# B&R Automation Studio project CControl_Gschneitner (part 5)

#### fbLascoSrvcInterv.st - Funktionsbaustein für Serviceintervalle
```iecst
(********************************************************************
 * COPYRIGHT -- LASCO Heu- und Forsttechnik GmbH
 ********************************************************************
 * Library: LascoUtil
 * Datei: fbLascoSrvcInterv.st
 * Autor: Rudolf Lachner
 * Erstellt: 16. Januar 2014
 ********************************************************************
 * Implementierung der Library LascoUtil
 ********************************************************************)

(* Funktionsbaustein für Serviceintervalle *)
FUNCTION_BLOCK fbLascoSrvcInterv

	//Service rücksetzen
	IF (EDGEPOS(SrvcReset)) THEN
		ZeitBisSrvc	:= SrvcIntervall;
	END_IF

	//Restzeit Countdown
	IF (Aktiv AND Tick) AND (ZeitBisSrvc > 0) THEN
		ZeitBisSrvc	:= ZeitBisSrvc - 1;
	END_IF

	//Service erforderlich
	IF (ZeitBisSrvc = 0) THEN
		SrvcErforderl	:= TRUE;
	ELSE
		SrvcErforderl	:= FALSE;
	END_IF

END_FUNCTION_BLOCK
```

#### fbLascoLstRamp.st - Rampenfunktion, Leistungsanstieg pro Minute
```iecst
(********************************************************************
 * COPYRIGHT -- LASCO Heu- und Forsttechnik GmbH
 ********************************************************************
 * Library: LascoUtil
 * Datei: fbLascoLstRamp.st
 * Autor: Rudolf Lachner
 * Erstellt: 21. Januar 2014
 ********************************************************************
 * Implementierung der Library LascoUtil
 ********************************************************************)

(* Rampenfunktion, Leistungsanstieg pro Minute *)
FUNCTION_BLOCK fbLascoLstRamp

	IF (EDGE(Enable)) THEN
		Fertig			:= FALSE;
		LeistungOut		:= LeistungStart;

	ELSIF (Enable AND sekTick) THEN

		AnstiegProSekunde	:= AnstiegProMinute / 60;

		IF ((LeistungOut + AnstiegProSekunde) <= LeistungSoll) AND NOT Pause THEN
			LeistungOut		:= LeistungOut + AnstiegProSekunde;
		ELSIF ((LeistungOut + AnstiegProSekunde) >= LeistungSoll) AND NOT Pause THEN
			IF LeistungSoll > LeistungStart THEN
				LeistungOut		:= LeistungSoll;
			ELSE
				LeistungOut		:= LeistungStart;
			END_IF
			Fertig 			:= TRUE;
		END_IF
	END_IF

END_FUNCTION_BLOCK
```

#### fbLascoBsk.st - Funktionsbaustein zur Ansteuerung von federrückgestellten Klappenantrieben
```iecst
(********************************************************************
 * COPYRIGHT -- LASCO Heu- und Forsttechnik GmbH
 ********************************************************************
 * Library: LascoUtil
 * Datei: fbLascoBsk.st
 * Autor: rlachner
 * Erstellt: 25. November 2014
 ********************************************************************
 * Implementierung der Library LascoUtil
 ********************************************************************)

(* Funktionsbaustein zur Ansteuerung von federrückgestellten Klappenantrieben *)
FUNCTION_BLOCK fbLascoBsk

	IF Freigabe THEN

		//Fahrzeiten überwachen
		TON_FahrzeitAuf(IN:= KlappeAuf AND NOT KlappeIstOffen AND NOT QuitFehler, PT:= FahrzeitAuf);
		TON_FahrzeitZu(IN:= NOT KlappeAuf AND NOT KlappeIstGeschlossen AND NOT QuitFehler, PT:= FahrzeitZu);

		FehlerFahrzeitAuf	:= TON_FahrzeitAuf.Q;
		FehlerFahrzeitZu	:= TON_FahrzeitZu.Q;

		//Stoerung Absicherung oder Endlagen
		IF (Stoerung) OR (KlappeIstOffen AND KlappeIstGeschlossen) THEN
			Fehler	:= TRUE;
		ELSE
			Fehler	:= FALSE;
		END_IF

		//Fehler rücksetzen
		IF (QuitFehler) THEN
			Fehler				:= FALSE;
		END_IF

		//Ansteuerung Klappe
		KlappeAuf	:= Oeffnen AND NOT Fehler;

	ELSE

		KlappeAuf			:= FALSE;
		Fehler				:= FALSE;
		FehlerFahrzeitAuf	:= FALSE;
		FehlerFahrzeitZu	:= FALSE;
		TON_FahrzeitAuf		(IN:= FALSE);
		TON_FahrzeitZu		(IN:= FALSE);

	END_IF

END_FUNCTION_BLOCK
```

#### fbLascoTrend.st - Trenderkennung eines Eingangswertes innerhalb einer Zeitspanne (steigend/fallend)
```iecst
(********************************************************************
 * COPYRIGHT -- LASCO Heu- und Forsttechnik GmbH
 ********************************************************************
 * Library: LascoUtil
 * Datei: fbLascoTrend.st
 * Autor: Rudolf Lachner
 * Erstellt: 3. Dezember 2014
 ********************************************************************
 * Implementierung der Library LascoUtil
 ********************************************************************)

(* Trenderkennung eines Eingangswertes innerhalb einer Zeitspanne (steigend/fallend) *)
FUNCTION_BLOCK fbLascoTrend

	IF (Freigabe AND (Zeitspanne <> 0)) THEN

		//Mittelwert neu berechnen
		IF (ctZeitspanne >= Zeitspanne) THEN

			Mittelwert	:= ((LREAL_TO_REAL(SummeWert)) / ctZeitspanne);

			//Berechnung der Abweichung
			IF Mittelwert - MittelwertMEM <> 0 THEN
				Abweichung := (((Mittelwert - MittelwertMEM) * 100 ) / ctZeitspanne);
			ELSE
				Abweichung := 0.0;
			END_IF

			//Steigende Tendenz erkannt
			IF MittelwertMEM < (Mittelwert - MinAbweichung) THEN
				TendenzSteigend := TRUE;
			ELSE
				TendenzSteigend := FALSE;
			END_IF

			//Fallende Tendenz erkannt
			IF MittelwertMEM > (Mittelwert + MinAbweichung) THEN
				TendenzFallend := TRUE;
			ELSE
				TendenzFallend := FALSE;
			END_IF

			MittelwertMEM	:= Mittelwert;
			ctZeitspanne	:= 0.0;
			SummeWert		:= 0.0;

		ELSIF Tick THEN

			SummeWert 		:=  SummeWert + Eingangswert;
			ctZeitspanne 	:= ctZeitspanne + 1;

		END_IF

	ELSE

		Abweichung		:= 0.0;
		ctZeitspanne	:= 0.0;
		Mittelwert		:= 0.0;
		MittelwertMEM	:= 0.0;
		SummeWert		:= 0.0;
		TendenzSteigend	:= FALSE;
		TendenzFallend	:= FALSE;

	END_IF

END_FUNCTION_BLOCK
```

#### fbLascoTimerHand.st - Timer mit Hand-Funktionen
```iecst
(********************************************************************
 * COPYRIGHT -- LASCO Heu- und Forsttechnik GmbH
 ********************************************************************
 * Library: LascoUtil
 * Datei: fbLascoTimerHand.st
 * Autor: Rudolf Lachner
 * Erstellt: 9. Dezember 2014
 ********************************************************************
 * Implementierung der Library LascoUtil
 ********************************************************************)

(* Timer mit Hand-Funktionen *)
FUNCTION_BLOCK fbLascoTimerHand

	IF (NOT Freigabe) THEN
		Elapsed	:= 0;
		Q		:= FALSE;
	ELSIF (HandEin) THEN
		Q		:= TRUE;
	ELSIF (HandAus) THEN
		Q		:= FALSE;
	ELSIF (Elapsed >= Zeit) THEN
		Q		:= FALSE;
	ELSE
		Elapsed	:= Elapsed + Tick;
		Q		:= TRUE;
	END_IF

END_FUNCTION_BLOCK
```

#### fbLascoBskUeberw.st - Ansteuerung Brandschutzklappe mit Laufzeitüberwachung und Freiräumung
```iecst
(********************************************************************
 * COPYRIGHT -- Lasco Heutechnik GmbH
 ********************************************************************
 * Library: LascoUtil
 * Datei: fbLascoBskUeberw.st
 * Autor: Rudolf Lachner
 * Erstellt: 20. Juli 2017
 ********************************************************************
 * Implementierung der Library LascoUtil
 ********************************************************************)

(* Ansteuerung Brandschutzklappe mit Laufzeitüberwachung und Freiräumung *)
FUNCTION_BLOCK fbLascoBskUeberw

	//Freigabe
	IF Freigabe THEN

		curStep	:= nextStep;

		//Schrittschaltwerk Überwachung Brandschutzklappe
		//***********************************************

		CASE curStep OF

			//*************************************************************************************************************************************************************************************************************************************
			BSK_WARTEN:

				//*** state entry ***
				IF stateEntry THEN
					stateEntry	:= FALSE;
					TON_Laufzeit(IN	:= FALSE, PT := T#0s);
				END_IF

				//*** state during ***
				//Warten auf Anforderung öffnen oder schließen

				//Fehlerquittierung
				IF Quit THEN
					ctVersucheAuf	:= 0;
					ctVersucheZu	:= 0;
				END_IF

				//*** state exit ***
				//Anforderung Öffnen
				IF FreigabeOeffnen AND NOT loc_KlappeIstOffen THEN
					stateEntry			:= TRUE;
					TON_Laufzeit(IN		:= FALSE, PT := T#0s);
					lastStep			:= curStep;
					nextStep			:= BSK_OEFFNEN;
				//Anforderung Schließen
				ELSIF FreigabeSchliessen AND NOT loc_KlappeIstGeschlossen THEN
					stateEntry			:= TRUE;
					TON_Laufzeit(IN		:= FALSE, PT := T#0s);
					lastStep			:= curStep;
					nextStep			:= BSK_SCHLIESSEN;
				END_IF

			//*************************************************************************************************************************************************************************************************************************************
			BSK_OEFFNEN:

				//*** state entry ***
				IF stateEntry THEN
					stateEntry					:= FALSE;
					TON_Laufzeit(IN				:= FALSE, PT := T#0s);
					loc_KlappeIstGeschlossen	:= FALSE;
					loc_KlappeIstOffen			:= FALSE;
					doKlappeOeffnen				:= TRUE;
				END_IF

				//*** state during ***

				//Laufzeit überwachen
				TON_Laufzeit(IN:= TRUE, PT := LaufzeitAuf);

				//*** state exit ***

				//Klappe ist offen
				IF diKlappeGeoeffnet AND NOT TON_Laufzeit.Q THEN
					TON_Laufzeit(IN		:= FALSE, PT := T#0s);
					ctVersucheAuf		:= 0;
					stateEntry			:= TRUE;
					lastStep			:= curStep;
					nextStep			:= BSK_WARTEN;
					loc_KlappeIstOffen	:= TRUE;

				//Laufzeitüberwachung ausggelöst
				ELSIF TON_Laufzeit.Q THEN
					//Max. Versuche überschritten -> Fehler
					IF ctVersucheAuf >= MaxVersucheAuf THEN
						TON_Laufzeit(IN		:= FALSE, PT := T#0s);
						stateEntry			:= TRUE;
						ctVersucheAuf		:= 0;
						lastStep			:= curStep;
						doKlappeOeffnen		:= FALSE;
						nextStep			:= BSK_STOERUNG;
					//Nächsten Versuch starten
					ELSE
						TON_Laufzeit(IN		:= FALSE, PT := T#0s);
						stateEntry			:= TRUE;
						ctVersucheAuf		:= ctVersucheAuf + 1;
						lastStep			:= curStep;
						doKlappeOeffnen		:= FALSE;
						nextStep			:= BSK_OEFFNEN_FEHLER;
					END_IF
				//Keine Anforderung
				ELSIF NOT FreigabeOeffnen THEN
					TON_Laufzeit(IN			:= FALSE, PT := T#0s);
					ctVersucheAuf			:= 0;
					stateEntry				:= TRUE;
					lastStep				:= curStep;
					nextStep				:= BSK_WARTEN;
				END_IF

			//*************************************************************************************************************************************************************************************************************************************
			BSK_OEFFNEN_FEHLER:

				//*** state entry ***
				IF stateEntry THEN
					stateEntry			:= FALSE;
					TON_Laufzeit(IN		:= FALSE, PT := T#0s);
				END_IF

				//*** state during ***

				//Laufzeit überwachen
				TON_Laufzeit(IN:= TRUE, PT := LaufzeitZu);

				//*** state exit ***
				//Klappe geschlossen -> Versuch öffnen
				IF diKlappeGeschlossen AND FreigabeOeffnen THEN
					stateEntry			:= TRUE;
					ctVersucheZu		:= 0;
					lastStep			:= curStep;
					nextStep			:= BSK_OEFFNEN;
					TON_Laufzeit(IN		:= FALSE, PT := T#0s);
				//Laufzeit überschritten
				ELSIF TON_Laufzeit.Q THEN
					//Max. Versuche überschritten -> Fehler
					IF ctVersucheZu >= MaxVersucheZu THEN
						TON_Laufzeit(IN		:= FALSE, PT := T#0s);
						stateEntry			:= TRUE;
						ctVersucheZu		:= 0;
						lastStep			:= curStep;
						doKlappeOeffnen		:= FALSE;
						nextStep			:= BSK_STOERUNG;
					//Nächsten Versuch starten
					ELSE
						TON_Laufzeit(IN		:= FALSE, PT := T#0s);
						stateEntry			:= TRUE;
						ctVersucheZu		:= ctVersucheZu + 1;
						lastStep			:= curStep;
						nextStep			:= BSK_OEFFNEN;
					END_IF
				//Keine Freigabe Öffnen
				ELSIF NOT FreigabeOeffnen THEN
					stateEntry				:= TRUE;
					TON_Laufzeit(IN			:= FALSE, PT := T#0s);
					lastStep				:= curStep;
					ctVersucheAuf			:= 0;
					nextStep				:= BSK_WARTEN;
				END_IF

			//*************************************************************************************************************************************************************************************************************************************
			BSK_SCHLIESSEN:

				//*** state entry ***
				IF stateEntry THEN
					stateEntry					:= FALSE;
					TON_Laufzeit(IN				:= FALSE, PT := T#0s);
					loc_KlappeIstGeschlossen	:= FALSE;
					loc_KlappeIstOffen			:= FALSE;
					doKlappeOeffnen				:= FALSE;
				END_IF

				//*** state during ***

				//Laufzeit überwachen
				TON_Laufzeit(IN:= TRUE, PT := LaufzeitZu);

				//*** state exit ***

				//Klappe ist geschlossen
				IF diKlappeGeschlossen AND NOT TON_Laufzeit.Q THEN
					TON_Laufzeit(IN				:= FALSE, PT := T#0s);
					ctVersucheZu				:= 0;
					stateEntry					:= TRUE;
					lastStep					:= curStep;
					nextStep					:= BSK_WARTEN;
					loc_KlappeIstGeschlossen	:= TRUE;

					//Laufzeitüberwachung ausgelöst
				ELSIF TON_Laufzeit.Q THEN
					//Max. Versuche überschritten -> Fehler
					IF ctVersucheZu >= MaxVersucheZu THEN
						TON_Laufzeit(IN		:= FALSE, PT := T#0s);
						stateEntry			:= TRUE;
						ctVersucheZu		:= 0;
						lastStep			:= curStep;
						doKlappeOeffnen		:= FALSE;
						nextStep			:= BSK_STOERUNG;
					//Nächsten Versuch starten
					ELSE
						TON_Laufzeit(IN		:= FALSE, PT := T#0s);
						stateEntry			:= TRUE;
						ctVersucheZu		:= ctVersucheZu + 1;
						lastStep			:= curStep;
						nextStep			:= BSK_SCHLIESSEN_FEHLER;
					END_IF
				//Anforderung Oeffnen
				ELSIF  FreigabeOeffnen THEN
					TON_Laufzeit(IN			:= FALSE, PT := T#0s);
					ctVersucheZu			:= 0;
					stateEntry				:= TRUE;
					lastStep				:= curStep;
					nextStep				:= BSK_WARTEN;
				END_IF

			//*************************************************************************************************************************************************************************************************************************************
			BSK_SCHLIESSEN_FEHLER:

				//*** state entry ***
				IF stateEntry THEN
					stateEntry			:= FALSE;
					TON_Laufzeit(IN		:= FALSE, PT := T#0s);
					doKlappeOeffnen		:= TRUE;
				END_IF

				//*** state during ***

				//Laufzeit überwachen
				TON_Laufzeit(IN:= TRUE, PT := LaufzeitAuf);

				//*** state exit ***
				//Klappe offen -> Versuch schließen
				IF diKlappeGeoeffnet AND FreigabeSchliessen THEN
					stateEntry			:= TRUE;
					ctVersucheAuf		:= 0;
					lastStep			:= curStep;
					nextStep			:= BSK_SCHLIESSEN;
					TON_Laufzeit(IN		:= FALSE, PT := T#0s);
				//Laufzeit überschritten
				ELSIF TON_Laufzeit.Q THEN
					//Max. Versuche überschritten -> Fehler
					IF ctVersucheAuf >= MaxVersucheAuf THEN
						TON_Laufzeit(IN		:= FALSE, PT := T#0s);
						stateEntry			:= TRUE;
						ctVersucheAuf		:= 0;
						lastStep			:= curStep;
						doKlappeOeffnen		:= FALSE;
						nextStep			:= BSK_STOERUNG;
						//Nächsten Versuch starten
					ELSE
						TON_Laufzeit(IN		:= FALSE, PT := T#0s);
						stateEntry			:= TRUE;
						ctVersucheAuf		:= ctVersucheAuf + 1;
						lastStep			:= curStep;
						nextStep			:= BSK_SCHLIESSEN;
					END_IF
					//Freigabe Öffnen
				ELSIF FreigabeOeffnen THEN
					stateEntry				:= TRUE;
					TON_Laufzeit(IN			:= FALSE, PT := T#0s);
					lastStep				:= curStep;
					ctVersucheZu			:= 0;
					nextStep				:= BSK_WARTEN;
				END_IF

			//*************************************************************************************************************************************************************************************************************************************
			BSK_STOERUNG:

				//*** state entry ***
				IF stateEntry THEN
					stateEntry		:= FALSE;
					TON_Laufzeit(IN	:= FALSE, PT := T#0s);
					Stoerung		:= TRUE;
				END_IF

				//*** state during ***
				//Warten auf Quittierung

				//*** state exit ***
				IF Quit THEN
					stateEntry	:= TRUE;
					Stoerung	:= FALSE;
					lastStep	:= curStep;
					nextStep	:= BSK_WARTEN;
				END_IF

		END_CASE

	//Keine Freigabe Funktionsbaustein
	ELSE

		//Alle Parameter zurücksetzen
		doKlappeOeffnen	:= FALSE;
		ctVersucheAuf	:= 0;
		ctVersucheZu	:= 0;
		Stoerung		:= FALSE;
		TON_Laufzeit(IN	:= FALSE, PT := T#0s);
		stateEntry		:= TRUE;
		curStep			:= BSK_WARTEN;
		nextStep		:= BSK_WARTEN;
		lastStep		:= BSK_WARTEN;

	END_IF

END_FUNCTION_BLOCK
```

#### fbLascoAutoRuecklauf.st - Automatische Rücklauffunktion für Motoren
```iecst
(********************************************************************
 * COPYRIGHT -- LASCO Heu- und Forsttechnik GmbH
 ********************************************************************
 * Library: LascoUtil
 * Datei: fbLascoAutoRuecklauf.st
 * Autor: rlachner
 * Erstellt: 24. Februar 2014
 ********************************************************************
 * Implementierung der Library LascoUtil
 ********************************************************************)

(* Automatische Rücklauffunktion für Motoren *)
FUNCTION_BLOCK fbLascoAutoRuecklauf

	IF Freigabe THEN

		CASE loc_curStep OF

			//AUS ********************************************************************************************************
			0:

				IF stateEntry THEN
					stateEntry := FALSE;
				END_IF

				MotorVor	:= FALSE;
				MotorRueck	:= FALSE;

				IF Zuendphase THEN
					stateEntry		:= TRUE;
					loc_curStep		:= 1;
				ELSIF Heizphase THEN
					stateEntry		:= TRUE;
					loc_curStep		:= 3;
				END_IF

			//ZUENDPHASE ***************************************************************************************************
			1:

				IF stateEntry THEN
					stateEntry 				:= FALSE;
					ctLaufzeitEinschub1		:= 0;
					ctLaufzeitEinschubVor	:= 0;
				END_IF

				MotorVor				:= (LaufzeitEinschubZuendung >= ctLaufzeitEinschub1);

				//Gesamtlaufzeit Motor Vor
				IF (ctLaufzeitEinschub1 <= LaufzeitEinschubZuendung) THEN
					ctLaufzeitEinschub1	:= ctLaufzeitEinschub1 + sekTick;
				END_IF

				//Laufzeit Vor am Stück
				IF MotorVor THEN
					ctLaufzeitEinschubVor	:= ctLaufzeitEinschubVor + sekTick;
				END_IF

				//Rücklauf erforderlich
				IF (ctLaufzeitEinschubVor >= MaxLaufzeitVor) AND (ctLaufzeitEinschub1 < LaufzeitEinschubZuendung) THEN
					loc_RuecklaufErforderlich	:= TRUE;
				END_IF

				//*** state exit ***
				IF (NOT Zuendphase) THEN
					stateEntry	:= TRUE;
					loc_curStep	:= 0;
				ELSIF loc_RuecklaufErforderlich THEN
					ctLaufzeitEinschubVor	:= 0;
					stateEntry	:= TRUE;
					loc_curStep	:= 2;
				END_IF

			//Zuendphase= Motor zurück ************************************************************************************************************
			2:

				IF stateEntry THEN
					stateEntry 				:= FALSE;
					MotorVor				:= FALSE;
					TON_Umschaltverz.IN		:= TRUE;
				END_IF

				TON_Umschaltverz.PT			:= VerzUmschaltung;
				TON_Umschaltverz();

				TOF_Ruecklauf.IN			:= TON_Umschaltverz.Q AND loc_RuecklaufErforderlich;
				TOF_Ruecklauf.PT			:= Ruecklaufzeit;
				TOF_Ruecklauf();

				MotorRueck					:= TOF_Ruecklauf.Q;

				IF MotorRueck THEN
					loc_RuecklaufErforderlich	:= FALSE;
				END_IF

				IF EDGENEG(MotorRueck) THEN
					loc_RueckwaertsOk	:= TRUE;
					TON_Umschaltverz(IN:= FALSE);
					TON_Umschaltverz.IN	:= TRUE;
				END_IF

				IF TON_Umschaltverz.Q AND loc_RueckwaertsOk THEN
					loc_RueckwaertsOk	:= FALSE;
					loc_curStep	:= 1;
					TON_Umschaltverz(IN:= FALSE);
					TOF_Ruecklauf(IN:= FALSE);
				ELSIF NOT Zuendphase THEN
					loc_curStep	:= 0;
					stateEntry	:= TRUE;
				END_IF

			//Heizphase ************************************************************************************************************
			3:

				//Vorwärts- Impulse mitzählen
				IF (EDGEPOS(ImpulsVor)) THEN
					ctEinschuebeSeitRuecklauf	:= ctEinschuebeSeitRuecklauf + 1;
				ELSIF (MotorRueck) THEN
					ctEinschuebeSeitRuecklauf	:= 0;
				END_IF

				//Kommando Rückwärtsfahrt erforderlich
				IF (ctEinschuebeSeitRuecklauf >= ImpulseVorBisRueck) AND NOT (ImpulsVor) THEN
					loc_RuecklaufErforderlich	:= TRUE;
				ELSIF (MotorRueck) THEN
					loc_RuecklaufErforderlich	:= FALSE;
				END_IF

				//Umschaltverzögerung
				IF (EDGENEG(ImpulsVor)) AND (loc_RuecklaufErforderlich) THEN
					TON_Umschaltverz.IN			:= TRUE;
				ELSIF (EDGEPOS(ImpulsVor)) THEN
					TON_Umschaltverz.IN			:= FALSE;
				END_IF

				//Rücklaufzeit
				TOF_Ruecklauf.IN	:= loc_RuecklaufErforderlich AND TON_Umschaltverz.Q;

				//Kommando "Motor Rückwärts"
				MotorRueck			:= TOF_Ruecklauf.Q;

				//Timer aufrufen
				TON_Umschaltverz.PT	:= UDINT_TO_TIME(VerzUmschaltung);
				TON_Umschaltverz();

				TOF_Ruecklauf.PT	:= UDINT_TO_TIME(Ruecklaufzeit);
				TOF_Ruecklauf();

				IF (NOT Heizphase) THEN
					loc_curStep	:= 0;
					stateEntry	:= TRUE;
				END_IF

		END_CASE

	ELSE

		stateEntry					:= TRUE;
		loc_curStep					:= 0;
		ctLaufzeitEinschub1			:= 0;
		ctLaufzeitEinschubVor		:= 0;
		MotorVor					:= FALSE;
		MotorRueck					:= FALSE;
		loc_RuecklaufErforderlich	:= FALSE;
		loc_RueckwaertsOk			:= FALSE;
		ctEinschuebeSeitRuecklauf	:= 0;
		TON_Umschaltverz.IN			:= FALSE;
		TOF_Ruecklauf.IN			:= FALSE;

	END_IF

END_FUNCTION_BLOCK
```

#### fbLascoPugeV2.st
```iecst
(* Puls/Pause-Generator mit Standard-Timern *)
FUNCTION_BLOCK fbLascoPugeV2

	curStep	:= nextStep;

	CASE curStep OF

		//*******************************************************************************************************************************************************************************
		0://WARTEN

			//*** state entry ***
			IF stateEntry THEN
				stateEntry := FALSE;
				PulsOut := FALSE;
				PauseOut := FALSE;
				TON_Schrittzeit(IN:= FALSE);
				RestzeitPause	:= 0;
				RestzeitPuls	:= 0;
			END_IF

			//*** state during ***

			//*** state exit ***
			IF (StartMitPuls) AND (ZeitPuls <> 0) THEN
				stateEntry := TRUE;
				nextStep	:= 2;
			ELSIF (StartMitPause) THEN
				stateEntry := TRUE;
				nextStep	:= 1;
			END_IF

			//***********************************************************************************************************************************************************************************
		1://PAUSE

			//*** state entry ***
			IF stateEntry THEN
				stateEntry := FALSE;
				PulsOut := FALSE;
				PauseOut := TRUE;
				TON_Schrittzeit(IN:= FALSE);
				RestzeitPause	:= 0;
				RestzeitPuls	:= 0;
			END_IF

			//*** state during ***
			TON_Schrittzeit(IN:= TRUE, PT:= UDINT_TO_TIME(ZeitPause));
			RestzeitPause := ZeitPause - TIME_TO_UDINT(TON_Schrittzeit.ET);

			//*** state exit ***
			IF (NOT StartMitPause AND NOT StartMitPuls) OR (ZeitPuls = 0) THEN
				stateEntry := TRUE;
				nextStep := 0;
			ELSIF TON_Schrittzeit.Q THEN
				stateEntry := TRUE;
				nextStep := 2;
			END_IF

			//************************************************************************************************************************************************************************************************
		2://PULS

			//*** state entry ***
			IF stateEntry THEN
				stateEntry := FALSE;
				PulsOut := TRUE;
				PauseOut := FALSE;
				TON_Schrittzeit(IN:= FALSE);
				RestzeitPause	:= 0;
				RestzeitPuls	:= 0;
			END_IF

			//*** state during ***
			TON_Schrittzeit(IN:= TRUE, PT:= UDINT_TO_TIME(ZeitPuls));
			RestzeitPuls := ZeitPuls - TIME_TO_UDINT(TON_Schrittzeit.ET);

			//*** state exit ***
			IF (NOT StartMitPause AND NOT StartMitPuls) OR (ZeitPuls = 0) THEN
				stateEntry := TRUE;
				nextStep := 0;
			ELSIF TON_Schrittzeit.Q THEN
				stateEntry := TRUE;
				nextStep := 1;
			END_IF

	END_CASE

END_FUNCTION_BLOCK
```

### Library Logical/Libraries/LaEntfV2 (IEC, version 1.00.0) - Funktionsblöcke für Entfeuchter ab LaTronicCControl407Plus

#### LaEntfV2.fun - Exported functions and function blocks
```iecst
{REDUND_UNREPLICABLE} FUNCTION_BLOCK fbEntfOelsumpfheiz (*Funktionsbaustein für Ansteuerung Ölsumpfheizung*) (*$GROUP=User,$CAT=User,$GROUPICON=User.png,$CATICON=User.png*)
	VAR_INPUT
		EintrittTemp : {REDUND_UNREPLICABLE} REAL;
		parTempOelsumpfheizungAus : {REDUND_UNREPLICABLE} REAL;
		parTempOelsumpfheizungEin : {REDUND_UNREPLICABLE} REAL;
		Freigabe : {REDUND_UNREPLICABLE} BOOL;
		StatusSensorEintrittOk : {REDUND_UNREPLICABLE} BOOL;
	END_VAR
	VAR_OUTPUT
		OelsumpfheizungEin : {REDUND_UNREPLICABLE} BOOL;
	END_VAR
END_FUNCTION_BLOCK

{REDUND_UNREPLICABLE} FUNCTION_BLOCK fbEntfKompressor (*Funktionsbaustein für Ansteuerung Kompressor*) (*$GROUP=User,$CAT=User,$GROUPICON=User.png,$CATICON=User.png*)
	VAR_INPUT
		EintrittFeuchte : {REDUND_UNREPLICABLE} REAL;
		SicherheitOk : {REDUND_UNREPLICABLE} BOOL;
		Freigabe : {REDUND_UNREPLICABLE} BOOL;
		BetriebsmldgVentilator : {REDUND_UNREPLICABLE} BOOL;
		Automatik : {REDUND_UNREPLICABLE} BOOL;
		Dauerbetrieb : {REDUND_UNREPLICABLE} BOOL;
		parFeuchteEin : {REDUND_UNREPLICABLE} REAL;
		parFeuchteAus : {REDUND_UNREPLICABLE} REAL;
		parEinschaltverzAbtau : {REDUND_UNREPLICABLE} UDINT;
		parAusschaltverzAbtau : {REDUND_UNREPLICABLE} UDINT;
		parEinschaltverzKompressor : {REDUND_UNREPLICABLE} UDINT;
		Hochdruck : {REDUND_UNREPLICABLE} REAL;
		Niederdruck : {REDUND_UNREPLICABLE} REAL;
		parNiederdruckMin : {REDUND_UNREPLICABLE} REAL;
		parHochdruckMax : {REDUND_UNREPLICABLE} REAL;
		parNiederdruckMax : {REDUND_UNREPLICABLE} REAL;
		StatusSensorNiederdruckOk : {REDUND_UNREPLICABLE} BOOL;
		StatusSensorEintrittOk : {REDUND_UNREPLICABLE} BOOL;
		DrehzahlvorgabeFU : {REDUND_UNREPLICABLE} REAL;
		BetriebsmldgKompressor : {REDUND_UNREPLICABLE} BOOL;
		DrehzahlMin : {REDUND_UNREPLICABLE} REAL;
		DrehzahlMax : {REDUND_UNREPLICABLE} REAL;
		RampeUp : {REDUND_UNREPLICABLE} REAL;
		RampeDown : {REDUND_UNREPLICABLE} REAL;
		QuitFehler : {REDUND_UNREPLICABLE} BOOL;
		parEinschaltverzMagnetventil : {REDUND_UNREPLICABLE} UDINT;
		parNiederdruckPumpdown : {REDUND_UNREPLICABLE} REAL;
		diNiederdruckOk : {REDUND_UNREPLICABLE} BOOL;
		diHochdruckOk : {REDUND_UNREPLICABLE} BOOL;
		KlappenumschaltungAkiv : {REDUND_UNREPLICABLE} BOOL;
		parVerzStandbyBeiKlappenumsch : {REDUND_UNREPLICABLE} UDINT;
	END_VAR
	VAR_OUTPUT
		FreigabeKompressorOut : {REDUND_UNREPLICABLE} BOOL;
		StoerungOut : {REDUND_UNREPLICABLE} BOOL;
		AbtauungAktiv : {REDUND_UNREPLICABLE} BOOL;
		DrehzahlOut : {REDUND_UNREPLICABLE} REAL;
		MagnetventilOut : {REDUND_UNREPLICABLE} BOOL;
		curStep : {REDUND_UNREPLICABLE} USINT;
		loc_StatusFeuchteOk : {REDUND_UNREPLICABLE} BOOL;
		FehlerPumpdown : {REDUND_UNREPLICABLE} BOOL;
		StandbyKlappenumsch : {REDUND_UNREPLICABLE} BOOL;
	END_VAR
	VAR
		TON_Abtau : {REDUND_UNREPLICABLE} TON;
		TON_Kompressor : {REDUND_UNREPLICABLE} TON;
		lastStep : {REDUND_UNREPLICABLE} USINT;
		nextStep : {REDUND_UNREPLICABLE} USINT;
		stateEntry : {REDUND_UNREPLICABLE} BOOL;
		fbFuKompressor : {REDUND_UNREPLICABLE} fbLascoFU;
		sekTick : {REDUND_UNREPLICABLE} BOOL;
		fbLascoEUhr_0 : {REDUND_UNREPLICABLE} fbLascoEUhr;
		fbLascoZdxx_0 : {REDUND_UNREPLICABLE} fbLascoZdxx;
		TON_EinschaltverzMagnetventil : {REDUND_UNREPLICABLE} TON;
		TON_LaufzeitPumpdown : {REDUND_UNREPLICABLE} TON;
		TON_Klappenumschaltung : {REDUND_UNREPLICABLE} TON;
	END_VAR
END_FUNCTION_BLOCK

{REDUND_ERROR} {REDUND_UNREPLICABLE} FUNCTION_BLOCK fbEntfFremd (*Funktionsbaustein zur Ansteuerung von Entfeuchtern (Fremdgeräte)*) (*$GROUP=User,$CAT=User,$GROUPICON=User.png,$CATICON=User.png*)
	VAR_INPUT
		Freigabe : {REDUND_UNREPLICABLE} BOOL;
		StoerungIn : {REDUND_UNREPLICABLE} BOOL;
		parVerzStoerung : {REDUND_UNREPLICABLE} UDINT;
		QuitFehler : {REDUND_UNREPLICABLE} BOOL;
		Dauerbetrieb : {REDUND_UNREPLICABLE} BOOL;
		Automatik : {REDUND_UNREPLICABLE} BOOL;
		BetriebsmldgVentilator : {REDUND_UNREPLICABLE} BOOL;
		parEinschaltverzKompressor : {REDUND_UNREPLICABLE} UDINT;
		BetriebsmldgEntfeuchter : {REDUND_UNREPLICABLE} BOOL;
		WitterungIstSchlecht : {REDUND_UNREPLICABLE} BOOL; (*Wenn TRUE, wird der Entfeuchter im Automatikbetrieb freigegeben*)
		parVerzBetriebEntfeuchter : {REDUND_UNREPLICABLE} UDINT;
	END_VAR
	VAR_OUTPUT
		StoerungOut : {REDUND_UNREPLICABLE} BOOL;
		FehlerBetriebsmldg : {REDUND_UNREPLICABLE} BOOL;
		FreigabeKompressorOut : {REDUND_UNREPLICABLE} BOOL;
	END_VAR
	VAR
		TON_Stoerung : {REDUND_UNREPLICABLE} TON;
		TON_VerzBetriebsmeldung : {REDUND_UNREPLICABLE} TON;
		curStep : {REDUND_UNREPLICABLE} USINT;
		nextStep : {REDUND_UNREPLICABLE} USINT;
		stateEntry : {REDUND_UNREPLICABLE} BOOL;
		TON_Kompressor : {REDUND_UNREPLICABLE} TON;
		lastStep : {REDUND_UNREPLICABLE} USINT;
	END_VAR
END_FUNCTION_BLOCK
```

#### fbEntfOelsumpfheiz.st
```iecst
(* Funktionsbaustein für Ansteuerung Oelsumpfheizung *)
FUNCTION_BLOCK fbEntfOelsumpfheiz

	//Ansteuerung Ölsumpfheizung
	//==========================

	IF Freigabe THEN

		OelsumpfheizungEin	:= TRUE;

	ELSE
		OelsumpfheizungEin	:= FALSE;
	END_IF

END_FUNCTION_BLOCK
```

#### fbEntfKompressor.st
```iecst
(* Ansteuerung Kompressor *)
FUNCTION_BLOCK fbEntfKompressor

	//Zeitticks erzeugen
	fbLascoEUhr_0(Freigabe := TRUE);
	fbLascoZdxx_0(IN := fbLascoEUhr_0.Sekunde);
	sekTick	:= fbLascoZdxx_0.Q;

	//Ausgang Störung Ein, wenn Sicherheitskreis nicht ok
	IF NOT SicherheitOk OR (fbFuKompressor.StoerungFU) THEN
		StoerungOut	:= TRUE;
	END_IF

	//Störung Laufzeit Pumpdown zurücksetzen, wenn Fehler quittiert
	IF QuitFehler THEN
		FehlerPumpdown	:= FALSE;
		StoerungOut		:= FALSE;
	END_IF

	//Funktionsbaustein FU Kompressor
	fbFuKompressor.AnsprechZeitFU	:= 5;
	fbFuKompressor.BetrMldg			:= BetriebsmldgKompressor;
	fbFuKompressor.MinDrehzahl		:= 0.0;
	fbFuKompressor.MaxDrehzahl		:= DrehzahlMax;
	fbFuKompressor.RampeUpSek		:= RampeUp;
	fbFuKompressor.RampeDownSek		:= RampeDown;
	fbFuKompressor.Reset			:= QuitFehler;
	fbFuKompressor.Tick				:= sekTick;
	fbFuKompressor();
	FreigabeKompressorOut			:= fbFuKompressor.BetriebFU;
	DrehzahlOut						:= fbFuKompressor.DrehzahlFU;

	//Schaltpunkte für Eintritt Feuchte generieren
	IF NOT Dauerbetrieb AND NOT Automatik THEN
		loc_StatusFeuchteOk := FALSE;
	ELSIF Dauerbetrieb THEN
		loc_StatusFeuchteOk	:= TRUE;
	ELSIF (EintrittFeuchte <= parFeuchteAus) AND loc_StatusFeuchteOk THEN
		loc_StatusFeuchteOk	:= FALSE;
	ELSIF (EintrittFeuchte >= parFeuchteEin) AND NOT loc_StatusFeuchteOk THEN
		loc_StatusFeuchteOk	:= TRUE;
	END_IF

	curStep	:= nextStep;

	CASE curStep OF

		//AUS **************************************************************************************************************************************
		0:

			//*** state entry ***
			IF stateEntry THEN
				stateEntry					:= FALSE;
				fbFuKompressor.Freigabe		:= FALSE;
				fbFuKompressor.SollDrehzahl	:= 0.0;
				TON_EinschaltverzMagnetventil(IN:= FALSE, PT:= 0);
				TON_Kompressor(IN:= FALSE, PT:= 0);
				TON_Abtau(IN:= FALSE, PT:= 0);
				AbtauungAktiv				:= FALSE;
				MagnetventilOut				:= FALSE;
			END_IF

			//*** state during ***
			//Warten auf Freigabe

			//*** state exit ***
			//Automatik oder Dauerbetrieb, Sensoren OK, Sicherheitskreis geschlossen, Ventilator in Betrieb -> Kompressor Ein
			IF ((Automatik AND StatusSensorEintrittOk) OR Dauerbetrieb) AND Freigabe AND StatusSensorNiederdruckOk AND loc_StatusFeuchteOk
				AND SicherheitOk AND BetriebsmldgVentilator AND diHochdruckOk AND diNiederdruckOk THEN
				nextStep	:= 1;
				lastStep	:= curStep;
				stateEntry	:= TRUE;
			ELSE
				nextStep	:= curStep;
			END_IF

		//KOMPRESSOR EIN **************************************************************************************************************************************
		1:

			//*** state entry ***
			IF stateEntry THEN
				stateEntry	:= FALSE;
				TON_Kompressor(IN:= FALSE, PT:= 0);
				fbFuKompressor.Freigabe		:= FALSE;
				fbFuKompressor.SollDrehzahl	:= 0.0;
				MagnetventilOut				:= FALSE;
				AbtauungAktiv				:= FALSE;
			END_IF

			//*** state during ***

			//Einschaltverzögerung Kompressor starten
			TON_Kompressor(IN:= TRUE, PT := parEinschaltverzKompressor);

			fbFuKompressor.Freigabe		:= TON_Kompressor.Q;
			fbFuKompressor.SollDrehzahl	:= DrehzahlvorgabeFU;

			//*** state exit ***
			//Keine Automatik und kein Dauerbetrieb, Sicherheit nicht ok, keine Betriebsmeldung Ventilator
			//oder Status Sensoren nicht ok -> AUS
			IF (NOT Automatik AND NOT Dauerbetrieb) OR (NOT StatusSensorEintrittOk AND Automatik) OR (NOT Freigabe) OR
				(NOT StatusSensorNiederdruckOk) OR (NOT SicherheitOk) OR (NOT BetriebsmldgVentilator) OR (NOT loc_StatusFeuchteOk) OR (NOT diHochdruckOk) OR (NOT diNiederdruckOk) THEN
				stateEntry	:= TRUE;
				lastStep	:= curStep;
				nextStep	:= 0;
			//Kompressor läuft -> Magnetventil Ein
			ELSIF fbFuKompressor.Freigabe THEN
				stateEntry	:= TRUE;
				lastStep	:= curStep;
				nextStep	:= 2;
			END_IF

		//MAGNETVENTIL EIN **************************************************************************************************************************************
		2:

			//*** state entry ***
			IF stateEntry THEN
				stateEntry	:= FALSE;
				TON_Kompressor(IN:= FALSE, PT:= 0);
				TON_EinschaltverzMagnetventil(IN:= FALSE, PT:= 0);
				MagnetventilOut				:= FALSE;
			END_IF

			//*** state during ***

			//Einschaltverzögerung Magnetventil
			TON_EinschaltverzMagnetventil(IN:= TRUE, PT:= parEinschaltverzMagnetventil);
			MagnetventilOut	:= (TON_EinschaltverzMagnetventil.Q) OR (parEinschaltverzMagnetventil = 0);

			//*** state exit ***
			//Keine Automatik und kein Dauerbetrieb, Sicherheit nicht ok, keine Betriebsmeldung Ventilator
			//oder Status Sensoren nicht ok -> Magnetventil Aus
			IF (NOT Automatik AND NOT Dauerbetrieb) OR (NOT StatusSensorEintrittOk AND Automatik) OR (NOT Freigabe) OR
				(NOT StatusSensorNiederdruckOk) OR (NOT SicherheitOk) OR (NOT BetriebsmldgVentilator) OR (NOT diHochdruckOk) OR (NOT diNiederdruckOk)  THEN
				stateEntry	:= TRUE;
				lastStep	:= curStep;
				IF MagnetventilOut THEN
					nextStep	:= 4;
				ELSE
					nextStep	:= 0;
				END_IF
			//Magnetventil Ein -> Betrieb
			ELSIF MagnetventilOut THEN
				stateEntry	:= TRUE;
				lastStep	:= curStep;
				nextStep	:= 3;
			END_IF

		//BETRIEB **************************************************************************************************************************************
		3:

			//*** state entry ***
			IF stateEntry THEN
				stateEntry		:= FALSE;
				TON_Abtau(IN:= FALSE, PT:= 0);
				AbtauungAktiv	:= FALSE;
				TON_Klappenumschaltung(IN:= FALSE, PT:= 0);
			END_IF

			//*** state during ***
			//Kompressor Drehzahlvorgabe
			fbFuKompressor.SollDrehzahl	:= DrehzahlvorgabeFU;

			//Verzöguerung Abtauung starten, wenn Niederdruck unter Min.
			TON_Abtau(IN:= (Niederdruck <= parNiederdruckMin), PT:= parEinschaltverzAbtau);

			//Wenn Hochdruck Max. überschritten & Klappenumschaltung aktiv -> Verzögerung starten für Standby
			TON_Klappenumschaltung(IN:= (Hochdruck > parHochdruckMax) AND KlappenumschaltungAkiv, PT:= parVerzStandbyBeiKlappenumsch);

			//*** state exit ***
			//Keine Automatik und kein Dauerbetrieb, Sicherheit nicht ok, keine Betriebsmeldung Ventilator
			//oder Status Sensoren nicht ok -> Magnetventil Aus
			IF (NOT Automatik AND NOT Dauerbetrieb) OR (NOT StatusSensorEintrittOk AND Automatik) OR (NOT Freigabe) OR
				(NOT StatusSensorNiederdruckOk) OR (NOT SicherheitOk) OR (NOT BetriebsmldgVentilator) OR (NOT loc_StatusFeuchteOk) OR (NOT diHochdruckOk) OR (NOT diNiederdruckOk) THEN
				stateEntry	:= TRUE;
				lastStep	:= curStep;
				nextStep	:= 4;
			//Abtauung angesprochen -> Abtauung
			ELSIF TON_Abtau.Q THEN
				stateEntry		:= TRUE;
				AbtauungAktiv	:= TRUE;
				nextStep		:= 6;
				lastStep		:= curStep;
			//Hochdruck Max. während Klappenumschaltung überschritten -> Standby
			ELSIF TON_Klappenumschaltung.Q THEN
				stateEntry		:= TRUE;
				nextStep		:= 7;
				lastStep		:= curStep;
			ELSE
				nextStep		:= curStep;
			END_IF

		//MAGNETVENTIL AUS **************************************************************************************************************************************
		4:

			//*** state entry ***
			IF stateEntry THEN
				stateEntry		:= FALSE;
				TON_Abtau(IN	:= FALSE, PT:= 0);
				AbtauungAktiv	:= FALSE;
				MagnetventilOut	:= FALSE;
				fbFuKompressor.SollDrehzahl	:= DrehzahlMin;
				TON_LaufzeitPumpdown(IN:= FALSE, PT:= 0);
			END_IF

			//*** state during ***

			//Laufzeit Pumpdown überwachen
			TON_LaufzeitPumpdown(IN:= TRUE, PT:= T#5m);

			//*** state exit ***
			//Automatik oder Dauerbetrieb, Sensoren und Sicherheit ok, Ventilator in Betrieb -> Betrieb
			IF ((Automatik AND StatusSensorEintrittOk) OR Dauerbetrieb) AND StatusSensorNiederdruckOk AND SicherheitOk AND Freigabe AND
				BetriebsmldgVentilator AND loc_StatusFeuchteOk THEN
				MagnetventilOut	:= TRUE;
				stateEntry	:= TRUE;
				lastStep	:= curStep;
				nextStep	:= 3;
			//Niederdruck < Pumpdown -> Kompressor Aus
			ELSIF (Niederdruck < parNiederdruckPumpdown) OR (NOT StatusSensorNiederdruckOk) OR fbFuKompressor.StoerungFU OR TON_LaufzeitPumpdown.Q OR (NOT diNiederdruckOk) OR (NOT diHochdruckOk) THEN
				stateEntry		:= TRUE;
				IF TON_LaufzeitPumpdown.Q THEN
					FehlerPumpdown	:= TRUE;
				END_IF
				TON_LaufzeitPumpdown(IN:= FALSE, PT:= 0);
				nextStep		:= 5;
				lastStep		:= curStep;
			ELSE
				nextStep		:= curStep;
			END_IF

		//KOMPRESSOR AUS **************************************************************************************************************************************
		5:

			//*** state entry ***
			IF stateEntry THEN
				stateEntry		:= FALSE;
				TON_Abtau(IN:= FALSE, PT:= 0);
				AbtauungAktiv	:= FALSE;
			END_IF

			//*** state during ***
			fbFuKompressor.Freigabe		:= FALSE;
			fbFuKompressor.SollDrehzahl	:= 0.0;

			//*** state exit ***
			//Kompressor Aus -> STILLSTAND
			stateEntry	:= TRUE;
			lastStep	:= curStep;
			nextStep	:= 0;

		//ABTAUUNG **************************************************************************************************************************************
		6:

			//*** state entry ***
			IF stateEntry THEN
				stateEntry		:= FALSE;
				TON_Abtau(IN:= FALSE, PT:= 0);
				AbtauungAktiv	:= TRUE;
				fbFuKompressor.SollDrehzahl	:= 0.0;
				MagnetventilOut	:= FALSE;
			END_IF

			//*** state during ***
			IF fbFuKompressor.DrehzahlFU = 0.0 THEN
				fbFuKompressor.Freigabe	:= FALSE;
			END_IF

			//Verzögerung Abtauung starten, wenn Niederdruck wieder über Min.
			TON_Abtau(IN:= (Niederdruck >= parNiederdruckMax), PT:= parAusschaltverzAbtau);

			//*** state exit ***
			//Keine Automatik und kein Dauerbetrieb, Sicherheit nicht ok, keine Betriebsmeldung Ventilator
			//oder Status Sensoren nicht ok -> Stillstand
			IF (NOT Automatik AND NOT Dauerbetrieb) OR (NOT StatusSensorEintrittOk AND Automatik) OR (NOT Freigabe) OR
				(NOT StatusSensorNiederdruckOk) OR (NOT SicherheitOk) OR (NOT BetriebsmldgVentilator) OR (NOT loc_StatusFeuchteOk) OR (NOT diHochdruckOk) OR (NOT diNiederdruckOk) THEN
				stateEntry	:= TRUE;
				lastStep	:= curStep;
				nextStep	:= 0;
			//Abtauung ok -> Kompressor Ein
			ELSIF TON_Abtau.Q THEN
				stateEntry	:= TRUE;
				lastStep	:= curStep;
				nextStep	:= 1;
			END_IF

		//STANDBY KLAPPENUMSCHALTUNG **************************************************************************************************************************************
		7:

			//*** state entry ***
			IF stateEntry THEN
				stateEntry		:= FALSE;
				TON_Klappenumschaltung(IN:= FALSE, PT:= 0);
				StandbyKlappenumsch	:= TRUE;
				fbFuKompressor.SollDrehzahl	:= 0.0;
				MagnetventilOut	:= FALSE;
			END_IF

			//*** state during ***
			IF fbFuKompressor.DrehzahlFU = 0.0 THEN
				fbFuKompressor.Freigabe	:= FALSE;
			END_IF

			//Verzögerung Ende Standby, wenn Klappenumschaltung abgeschlossen
			TON_Klappenumschaltung(IN:= NOT KlappenumschaltungAkiv, PT:= parVerzStandbyBeiKlappenumsch);

			//*** state exit ***
			//Keine Automatik und kein Dauerbetrieb, Sicherheit nicht ok, keine Betriebsmeldung Ventilator
			//oder Status Sensoren nicht ok -> Stillstand
			IF (NOT Automatik AND NOT Dauerbetrieb) OR (NOT StatusSensorEintrittOk AND Automatik) OR (NOT Freigabe) OR
				(NOT StatusSensorNiederdruckOk) OR (NOT SicherheitOk) OR (NOT BetriebsmldgVentilator) OR (NOT loc_StatusFeuchteOk) OR (NOT diHochdruckOk) OR (NOT diNiederdruckOk) THEN
				stateEntry	:= TRUE;
				StandbyKlappenumsch	:= FALSE;
				lastStep	:= curStep;
				nextStep	:= 0;
			//Klappenumschaltung abgeschlossen -> Kompressor Ein
			ELSIF TON_Klappenumschaltung.Q THEN
				stateEntry	:= TRUE;
				StandbyKlappenumsch	:= FALSE;
				lastStep	:= curStep;
				nextStep	:= 1;
			END_IF

	END_CASE

END_FUNCTION_BLOCK
```

#### fbEntfFremd.st
```iecst
(* Funktionsbaustein zur Ansteuerung von Entfeuchtern (Fremdgeräte) *)
FUNCTION_BLOCK fbEntfFremd

	//Ausgang Störung Ein, wenn Störmeldung von Entfeuchter
	TON_Stoerung(IN:= StoerungIn, PT:= parVerzStoerung);

	//Störungseingang oder keine Betriebsmeldung Entfeuchter nach Freigabe -> Störung generieren
	IF TON_Stoerung.Q OR TON_VerzBetriebsmeldung.Q THEN
		StoerungOut	:= TRUE;
	END_IF

	//Eigenen Fehlerausgang, wenn keine Betriebsmeldung von Entfeuchter (für Alarme)
	IF TON_VerzBetriebsmeldung.Q THEN
		FehlerBetriebsmldg := TRUE;
	END_IF

	//Störung zurücksetzen, wenn Fehler quittiert
	IF QuitFehler AND NOT StoerungIn THEN
		StoerungOut		:= FALSE;
		FehlerBetriebsmldg := FALSE;
	END_IF

	curStep	:= nextStep;

	CASE curStep OF

		//AUS **************************************************************************************************************************************
		0:

			//*** state entry ***
			IF stateEntry THEN
				stateEntry					:= FALSE;
				FreigabeKompressorOut		:= FALSE;
				TON_Kompressor(IN:= FALSE, PT:= 0);
				TON_VerzBetriebsmeldung(IN:= FALSE, PT:= 0);
			END_IF

			//*** state during ***
			//Warten auf Freigabe

			//*** state exit ***
			//Automatik oder Dauerbetrieb, Sensoren OK, keine Stoerung, Ventilator in Betrieb -> Kompressor Ein
			IF ((Automatik AND WitterungIstSchlecht) OR Dauerbetrieb) AND Freigabe AND BetriebsmldgVentilator AND NOT StoerungOut THEN
				nextStep	:= 1;
				lastStep	:= curStep;
				stateEntry	:= TRUE;
			ELSE
				nextStep	:= curStep;
			END_IF

			//ENTFEUCHTER EINSCHALTVERZÖGERUNG **************************************************************************************************************************************
		1:

			//*** state entry ***
			IF stateEntry THEN
				stateEntry	:= FALSE;
				TON_Kompressor(IN:= FALSE, PT:= 0);
				FreigabeKompressorOut		:= FALSE;
			END_IF

			//*** state during ***

			//Einschaltverzögerung Kompressor starten
			TON_Kompressor(IN:= TRUE, PT := parEinschaltverzKompressor);

			//*** state exit ***
			//Keine Automatik und kein Dauerbetrieb, Störung, keine Betriebsmeldung Ventilator
			//oder Status Sensoren nicht ok -> AUS
			IF (NOT Automatik AND NOT Dauerbetrieb) OR (NOT WitterungIstSchlecht AND Automatik) OR (NOT Freigabe) OR
				(StoerungOut) OR (NOT BetriebsmldgVentilator) THEN
				stateEntry	:= TRUE;
				lastStep	:= curStep;
				nextStep	:= 0;
				//Einschaltverzögerung abgelaufen -> Betrieb
			ELSIF TON_Kompressor.Q THEN
				stateEntry	:= TRUE;
				lastStep	:= curStep;
				nextStep	:= 2;
			END_IF

			//ENTFEUCHTER BETRIEB **************************************************************************************************************************************
		2:

			//*** state entry ***
			IF stateEntry THEN
				stateEntry	:= FALSE;
				TON_Kompressor(IN:= FALSE, PT:= 0);
				TON_VerzBetriebsmeldung(IN:= FALSE, PT:= 0);
			END_IF

			//*** state during ***

			//Entfeuchter freigeben
			FreigabeKompressorOut := TRUE;

			//Betriebsmeldung Entfeuchter verzögert abfragen
			TON_VerzBetriebsmeldung(IN:= FreigabeKompressorOut AND NOT BetriebsmldgEntfeuchter, PT:= parVerzBetriebEntfeuchter);

			//*** state exit ***
			//Keine Freigabe, Störung oder keine Betriebsmeldung Ventilator -> AUS
			IF (NOT Automatik AND NOT Dauerbetrieb) OR (NOT Freigabe) OR
				(NOT WitterungIstSchlecht AND Automatik) OR (StoerungOut) OR (NOT BetriebsmldgVentilator) THEN
				stateEntry := TRUE;
				lastStep := curStep;
				nextStep := 3;
			ELSE
				nextStep := curStep;
			END_IF

			//ENTFEUCHTER AUS **************************************************************************************************************************************
		3:

			//*** state entry ***
			IF stateEntry THEN
				stateEntry		:= FALSE;
				TON_Kompressor(IN:= FALSE, PT:= 0);
				TON_VerzBetriebsmeldung(IN:= FALSE, PT:= 0);
				FreigabeKompressorOut := FALSE;
			END_IF

			//*** state exit ***
			stateEntry := TRUE;
			lastStep := curStep;
			nextStep := 0;

	END_CASE

END_FUNCTION_BLOCK
```

### Library Logical/Libraries/LascoBoxen (IEC, version 1.00.0)

#### Types.typ - Exported data types
```iecst
TYPE
	typBoxenLuftmengenIn : {REDUND_UNREPLICABLE} 	STRUCT
		GrundflaecheBox : {REDUND_UNREPLICABLE} REAL;
		BoxIstAktiv : {REDUND_UNREPLICABLE} BOOL;
		Ventilator1 : {REDUND_UNREPLICABLE} BOOL;
		Ventilator2 : {REDUND_UNREPLICABLE} BOOL;
	END_STRUCT;
	typKonfigurationBoxenOut : {REDUND_UNREPLICABLE} 	STRUCT
		RestzeitSchlechtwetterPuls : {REDUND_UNREPLICABLE} UDINT; (*Restzeit Pulszeit Schlechtwetterbetrieb [ms]*)
		RestzeitSchlechtwetterPause : {REDUND_UNREPLICABLE} UDINT; (*Restzeit Pausezeit Schlechtwetterbetrieb [ms]*)
		BoxBereit : {REDUND_UNREPLICABLE} BOOL; (*Betriebsart Box <> AUS*)
		BoxAktiv : {REDUND_UNREPLICABLE} BOOL; (*Betriebsart Box <> AUS und Dauerbetrieb oder Zeitbereiche Intervall/Nachtrocknung sind aktiv*)
		DauerbetriebSperre : {REDUND_UNREPLICABLE} BOOL; (*Sperre von Dauerbetrieb für Box*)
		IntervallbetriebSperre : {REDUND_UNREPLICABLE} BOOL; (*Sperre von Intervallbetrieb für Box*)
		IntervallbetriebZeitenGesperrt : {REDUND_UNREPLICABLE} ARRAY[0..23]OF BOOL; (*Zeitfenster Intervallbetrieb gesperrt (weil von anderer Box im selben Lüfterkreis gewählt)*)
		NachtrocknungZeitenGesperrt : {REDUND_UNREPLICABLE} ARRAY[0..23]OF BOOL; (*Zeitfenster Nachtrocknung gesperrt (weil von anderer Box im selben Lüfterkreis gewählt)*)
	END_STRUCT;
	typKonfigurationBoxenIn : {REDUND_UNREPLICABLE} 	STRUCT
		Ventilator1 : {REDUND_UNREPLICABLE} BOOL; (*0= Box wird nicht über Ventilator 1 versorgt, 1= Box wird über Ventilator 1 versorgt*)
		Ventilator2 : {REDUND_UNREPLICABLE} BOOL; (*0= Box wird nicht über Ventilator 2 versorgt, 1= Box wird über Ventilator 2 versorgt*)
		Luftentfeuchter : {REDUND_UNREPLICABLE} BOOL; (*0= Luftentfeuchter nicht vorhanden oder nicht von Box verwendet, 1= Luftentfeuchter wird von Box verwendet*)
		Warmluftofen : {REDUND_UNREPLICABLE} BOOL; (*0= Warmluftofen nicht vorhanden oder nicht von Box verwendet, 1= Warmluftofen wird von Box verwendet*)
		Heizregister : {REDUND_UNREPLICABLE} BOOL; (*0= Heizregister nicht vorhanden oder nicht von Box verwendet, 1= Heizregister wird von Box verwendet*)
		Scheitholzofen : {REDUND_UNREPLICABLE} BOOL; (*0= Scheitholzofen nicht vorhanden oder nicht von Box verwendet, 1= Scheitholzofen wird von Box verwendet*)
		StellungKlappe1 : {REDUND_UNREPLICABLE} enumStellungKlappenBoxen; (*0= Klappe nicht vorhanden oder nicht von Box verwendet, 1= Klappe bei Ansteuerung der Box geschlossen, 2= Klappe bei Ansteuerung der Box geöffnet*)
		StellungKlappe2 : {REDUND_UNREPLICABLE} enumStellungKlappenBoxen; (*0= Klappe nicht vorhanden oder nicht von Box verwendet, 1= Klappe bei Ansteuerung der Box geschlossen, 2= Klappe bei Ansteuerung der Box geöffnet*)
		StellungKlappe3 : {REDUND_UNREPLICABLE} enumStellungKlappenBoxen; (*0= Klappe nicht vorhanden oder nicht von Box verwendet, 1= Klappe bei Ansteuerung der Box geschlossen, 2= Klappe bei Ansteuerung der Box geöffnet*)
		StellungKlappe4 : {REDUND_UNREPLICABLE} enumStellungKlappenBoxen; (*0= Klappe nicht vorhanden oder nicht von Box verwendet, 1= Klappe bei Ansteuerung der Box geschlossen, 2= Klappe bei Ansteuerung der Box geöffnet*)
		StellungKlappe5 : {REDUND_UNREPLICABLE} enumStellungKlappenBoxen; (*0= Klappe nicht vorhanden oder nicht von Box verwendet, 1= Klappe bei Ansteuerung der Box geschlossen, 2= Klappe bei Ansteuerung der Box geöffnet*)
		StellungKlappe6 : {REDUND_UNREPLICABLE} enumStellungKlappenBoxen; (*0= Klappe nicht vorhanden oder nicht von Box verwendet, 1= Klappe bei Ansteuerung der Box geschlossen, 2= Klappe bei Ansteuerung der Box geöffnet*)
		DauerbetriebEin : {REDUND_UNREPLICABLE} BOOL; (*Betriebsart Dauerbetrieb ausgewählt (Automatikbetrieb)*)
		WetterIstSchlecht : {REDUND_UNREPLICABLE} BOOL; (*Wenn TRUE, wird im Automatikbetrieb auf Puls/Pausebetrieb umgeschaltet, wenn keine Luftaufbereitung verfügbar ist.*)
		LuftaufbIstVerfuegbar : {REDUND_UNREPLICABLE} BOOL; (*TRUE, wenn eine Luftaufbereitung verfügbar ist (In Ausstattung vorhanden, Betriebsart <> AUS, kein Fehler)*)
		IntervallbetriebEin : {REDUND_UNREPLICABLE} BOOL; (*Betriebsart Intervallbetrieb ausgewählt*)
		NachtrocknungEin : {REDUND_UNREPLICABLE} BOOL; (*Betriebsart Nachtrocknung ausgewählt*)
		IntervallbetriebZeiten : {REDUND_UNREPLICABLE} ARRAY[0..23]OF BOOL; (*Zeitfenster Intervallbetrieb*)
		NachtrocknungZeiten : {REDUND_UNREPLICABLE} ARRAY[0..23]OF BOOL; (*Zeitfenster Nachtrocknung*)
		SchlechtwetterPulszeit : {REDUND_UNREPLICABLE} UDINT; (*Pulszeit bei Schlechtwettterbetrieb [ms]*)
		SchlechtwetterPausezeit : {REDUND_UNREPLICABLE} UDINT; (*Pausezeit bei Schlechtwetterbetrieb [ms]*)
	END_STRUCT;
	enumStellungKlappenBoxen :
		(
		FBBOX_NICHT_VERWENDET := 0, (*Stellung der Klappe für Box nicht relevant*)
		FBBOX_GESCHLOSSEN := 1,
		FBBOX_GEOEFFNET := 2
		);
END_TYPE
```

#### LascoBoxen.fun - Exported functions and function blocks
```iecst
{REDUND_ERROR} {REDUND_UNREPLICABLE} FUNCTION_BLOCK fbBoxenKonfig (*Funktionsbaustein für Konfiguration der einzelnen Boxen (Anforderung Box, Klappen, Ventilatoren, Luftaufbereitung,...)*) (*$GROUP=User,$CAT=User,$GROUPICON=User.png,$CATICON=User.png*)
	VAR_INPUT
		StundeAktuell : {REDUND_UNREPLICABLE} USINT; (*Aktuelle Stunde (0-23h)*)
		ScheitholzofenNochAktiv : {REDUND_UNREPLICABLE} BOOL; (*Für Notbetrieb Boxen und Ventilatoren, wenn Boxen in Pause oder Stillstand und Scheitholzofen noch aktiv*)
		EntfeuchterNochAktiv : {REDUND_UNREPLICABLE} BOOL; (*Für Notbetrieb Boxen und Ventilatoren, wenn Boxen in Pause oder Stillstand und Entfeuchter noch aktiv*)
		BypassklVonBeidenVentAbhaengig : {REDUND_UNREPLICABLE} BOOL; (*Wenn TRUE, werden beide Ventilatoren bei Umschaltung Bypassklappe auf Min-Drehzahl gefahren (wird an Baustein für Ventilatoren übergeben*)
		BoxenklVonBeidenVentAbhaengig : {REDUND_UNREPLICABLE} BOOL; (*Wenn TRUE, werden beide Ventilatoren bei Klappenumschaltung auf Min-Drehzahl gefahren (wird an Baustein für Ventilatoren übergeben*)
		WarmluftofenNochAktiv : {REDUND_UNREPLICABLE} BOOL; (*Für Notbetrieb Boxen und Ventilatoren, wenn Boxen in Pause oder Stillstand und Warmluftofen noch aktiv*)
		AlleKlappenSchliessenWennAus : {REDUND_UNREPLICABLE} BOOL; (*Wenn TRUE, werden alle Klappen geschlossen wenn keine Box im jeweiligen Lüfterkreis aktiv ist*)
		MehrereBoxenBelueftbar : {REDUND_UNREPLICABLE} BOOL; (*Wenn TRUE, können mehrere Boxen pro Lüfterkreis gleichzeitig belüftet werden (z.B. bei Anlagen mit Jalousieklappen)*)
		Box1In : {REDUND_UNREPLICABLE} typKonfigurationBoxenIn;
		Box2In : {REDUND_UNREPLICABLE} typKonfigurationBoxenIn;
		Box3In : {REDUND_UNREPLICABLE} typKonfigurationBoxenIn;
		Box4In : {REDUND_UNREPLICABLE} typKonfigurationBoxenIn;
		Box5In : {REDUND_UNREPLICABLE} typKonfigurationBoxenIn;
		Box6In : {REDUND_UNREPLICABLE} typKonfigurationBoxenIn;
		EntfeuchterInselbetrieb : {REDUND_UNREPLICABLE} BOOL; (*Für 3.04: Wenn kein Ventilator in Ausstattung ausgewählt, wird der Entfeuchter im Inselbetrieb (Start/Stopp über Extern) betrieben*)
		TasteEntfeuchterEinInselbetrieb : {REDUND_UNREPLICABLE} BOOL; (*Für 3.04: TRUE, wenn Taste "Entfeuchter freigeben" im Inselbetrieb eingeschaltet ist*)
		AnfEntfeuchterExtern : {REDUND_UNREPLICABLE} BOOL; (*Für 3.04, TRUE, wenn Entfeuchter wird über Fremdsteuerung angefordert wird*)
	END_VAR
	VAR_OUTPUT
		Box1Out : {REDUND_UNREPLICABLE} typKonfigurationBoxenOut;
		Box2Out : {REDUND_UNREPLICABLE} typKonfigurationBoxenOut;
		Box3Out : {REDUND_UNREPLICABLE} typKonfigurationBoxenOut;
		Box4Out : {REDUND_UNREPLICABLE} typKonfigurationBoxenOut;
		Box5Out : {REDUND_UNREPLICABLE} typKonfigurationBoxenOut;
		Box6Out : {REDUND_UNREPLICABLE} typKonfigurationBoxenOut;
		FreigabeKlappe1Out : {REDUND_UNREPLICABLE} BOOL;
		FreigabeKlappe2Out : {REDUND_UNREPLICABLE} BOOL;
		FreigabeKlappe3Out : {REDUND_UNREPLICABLE} BOOL;
		FreigabeKlappe4Out : {REDUND_UNREPLICABLE} BOOL;
		FreigabeKlappe5Out : {REDUND_UNREPLICABLE} BOOL;
		FreigabeKlappe6Out : {REDUND_UNREPLICABLE} BOOL;
		FreigabeVentilator1 : {REDUND_UNREPLICABLE} BOOL;
		FreigabeVentilator2 : {REDUND_UNREPLICABLE} BOOL;
		FreigabeLuftentfeuchter : {REDUND_UNREPLICABLE} BOOL;
		FreigabeWarmluftofen : {REDUND_UNREPLICABLE} BOOL;
		FreigabeHeizregister : {REDUND_UNREPLICABLE} BOOL;
		FreigabeScheitholzofen : {REDUND_UNREPLICABLE} BOOL;
		EntfeuchterVonVent1Abhaengig : {REDUND_UNREPLICABLE} BOOL; (*Wird freigegeben, wenn Entfeuchter von Ventilator 1 abhängig ist (damit Ventilator läuft, wenn Entfeuchter noch aktiv)*)
		EntfeuchterVonVent2Abhaengig : {REDUND_UNREPLICABLE} BOOL; (*Wird freigegeben, wenn Entfeuchter von Ventilator 2 abhängig ist (damit Ventilator läuft, wenn Entfeuchter aktiv)*)
		WarmluftofenVonVent1Abhaengig : {REDUND_UNREPLICABLE} BOOL; (*Wird freigegeben, wenn Warmluftofen von Ventilator 1 abhängig ist (damit Ventilator läuft, wenn Warmluftofen aktiv)*)
		WarmluftofenVonVent2Abhaengig : {REDUND_UNREPLICABLE} BOOL; (*Wird freigegeben, wenn Warmluftofen von Ventilator 2 abhängig ist (damit Ventilator läuft, wenn Warmluftofen aktiv)*)
		HeizregisterVonVent1Abhaengig : {REDUND_UNREPLICABLE} BOOL; (*Wird freigegeben, wenn Heizregister von Ventilator 1 abhängig ist (damit Ventilator läuft, wenn Heizregister aktiv)*)
		HeizregisterVonVent2Abhaengig : {REDUND_UNREPLICABLE} BOOL; (*Wird freigegeben, wenn Heizregister von Ventilator 2 abhängig ist (damit Ventilator läuft, wenn Heizregister aktiv)*)
		ScheitholzofenVonVent1Abhaengig : {REDUND_UNREPLICABLE} BOOL; (*Wird freigegeben, wenn Scheitholzofen von Ventilator 1 abhängig ist (damit Ventilator läuft, wenn Scheitholzofen aktiv)*)
		ScheitholzofenVonVent2Abhaengig : {REDUND_UNREPLICABLE} BOOL; (*Wird freigegeben, wenn Scheitholzofen von Ventilator 2 abhängig ist (damit Ventilator läuft, wenn Scheitholzofen aktiv)*)
		NotbetriebBox1 : {REDUND_UNREPLICABLE} BOOL;
		NotbetriebBox2 : {REDUND_UNREPLICABLE} BOOL;
		NotbetriebBox3 : {REDUND_UNREPLICABLE} BOOL;
		NotbetriebBox4 : {REDUND_UNREPLICABLE} BOOL;
		NotbetriebBox5 : {REDUND_UNREPLICABLE} BOOL;
		NotbetriebBox6 : {REDUND_UNREPLICABLE} BOOL;
		NotbetriebVentilator1 : {REDUND_UNREPLICABLE} BOOL; (*Freigabe für Notbetrieb Ventilator 1 (keine Box aktiv, jedoch Trocknungsgeräte noch im Nachlauf (Auskühlphasen Öfen)*)
		NotbetriebVentilator2 : {REDUND_UNREPLICABLE} BOOL; (*Freigabe für Notbetrieb Ventilator 2 (keine Box aktiv, jedoch Trocknungsgeräte noch im Nachlauf (Auskühlphasen Öfen)*)
		Boxenkl1VonVent1Abhaengig : {REDUND_UNREPLICABLE} BOOL; (*Wird an Baustein für Ansteuerung Ventilatoren übergeben (nur jeweiligen Ventilator bei Klappenumschaltung ausschalten)*)
		Boxenkl1VonVent2Abhaengig : {REDUND_UNREPLICABLE} BOOL; (*Wird an Baustein für Ansteuerung Ventilatoren übergeben (nur jeweiligen Ventilator bei Klappenumschaltung ausschalten)*)
		Boxenkl2VonVent1Abhaengig : {REDUND_UNREPLICABLE} BOOL; (*Wird an Baustein für Ansteuerung Ventilatoren übergeben (nur jeweiligen Ventilator bei Klappenumschaltung ausschalten)*)
		Boxenkl2VonVent2Abhaengig : {REDUND_UNREPLICABLE} BOOL; (*Wird an Baustein für Ansteuerung Ventilatoren übergeben (nur jeweiligen Ventilator bei Klappenumschaltung ausschalten)*)
		Boxenkl3VonVent1Abhaengig : {REDUND_UNREPLICABLE} BOOL; (*Wird an Baustein für Ansteuerung Ventilatoren übergeben (nur jeweiligen Ventilator bei Klappenumschaltung ausschalten)*)
		Boxenkl3VonVent2Abhaengig : {REDUND_UNREPLICABLE} BOOL; (*Wird an Baustein für Ansteuerung Ventilatoren übergeben (nur jeweiligen Ventilator bei Klappenumschaltung ausschalten)*)
		Boxenkl4VonVent1Abhaengig : {REDUND_UNREPLICABLE} BOOL; (*Wird an Baustein für Ansteuerung Ventilatoren übergeben (nur jeweiligen Ventilator bei Klappenumschaltung ausschalten)*)
		Boxenkl4VonVent2Abhaengig : {REDUND_UNREPLICABLE} BOOL; (*Wird an Baustein für Ansteuerung Ventilatoren übergeben (nur jeweiligen Ventilator bei Klappenumschaltung ausschalten)*)
		Boxenkl5VonVent1Abhaengig : {REDUND_UNREPLICABLE} BOOL; (*Wird an Baustein für Ansteuerung Ventilatoren übergeben (nur jeweiligen Ventilator bei Klappenumschaltung ausschalten)*)
		Boxenkl5VonVent2Abhaengig : {REDUND_UNREPLICABLE} BOOL; (*Wird an Baustein für Ansteuerung Ventilatoren übergeben (nur jeweiligen Ventilator bei Klappenumschaltung ausschalten)*)
		Boxenkl6VonVent1Abhaengig : {REDUND_UNREPLICABLE} BOOL; (*Wird an Baustein für Ansteuerung Ventilatoren übergeben (nur jeweiligen Ventilator bei Klappenumschaltung ausschalten)*)
		Boxenkl6VonVent2Abhaengig : {REDUND_UNREPLICABLE} BOOL; (*Wird an Baustein für Ansteuerung Ventilatoren übergeben (nur jeweiligen Ventilator bei Klappenumschaltung ausschalten)*)
		BypassklVonVent1Abhaengig : {REDUND_UNREPLICABLE} BOOL; (*Wird an Baustein für Ansteuerung Ventilatoren übergeben (nur jeweiligen Ventilator bei Klappenumschaltung ausschalten)*)
		BypassklVonVent2Abhaengig : {REDUND_UNREPLICABLE} BOOL; (*Wird an Baustein für Ansteuerung Ventilatoren übergeben (nur jeweiligen Ventilator bei Klappenumschaltung ausschalten)*)
		FreigabeEntfeuchterInselbetrieb : {REDUND_UNREPLICABLE} BOOL; (*Für 3.04: Freigabe Luftentfeuchter, wenn über Fremdsteuerung angefordert*)
		EntfeuchterInselbetrAktivOut : {REDUND_UNREPLICABLE} BOOL; (*TRUE, wenn Entfeuchter im Inselbetrieb betrieben wird & Taste "EIN" für Inselbetrieb aktiv ist.*)
	END_VAR
	VAR
		fbPugeSchlechtwetterBox1 : {REDUND_UNREPLICABLE} fbLascoPugeV2;
		fbPugeSchlechtwetterBox2 : {REDUND_UNREPLICABLE} fbLascoPugeV2;
		fbPugeSchlechtwetterBox3 : {REDUND_UNREPLICABLE} fbLascoPugeV2;
		fbPugeSchlechtwetterBox4 : {REDUND_UNREPLICABLE} fbLascoPugeV2;
		fbPugeSchlechtwetterBox5 : {REDUND_UNREPLICABLE} fbLascoPugeV2;
		fbPugeSchlechtwetterBox6 : {REDUND_UNREPLICABLE} fbLascoPugeV2;
		i : {REDUND_UNREPLICABLE} INT; (*Schleifenzähler*)
		loc_Box1GleicherLuefterkreis : {REDUND_UNREPLICABLE} BOOL;
		loc_Box2GleicherLuefterkreis : {REDUND_UNREPLICABLE} BOOL;
		loc_Box3GleicherLuefterkreis : {REDUND_UNREPLICABLE} BOOL;
		loc_Box4GleicherLuefterkreis : {REDUND_UNREPLICABLE} BOOL;
		loc_Box5GleicherLuefterkreis : {REDUND_UNREPLICABLE} BOOL;
		loc_Box6GleicherLuefterkreis : {REDUND_UNREPLICABLE} BOOL;
		loc_Entf_NotbetriebBox1 : {REDUND_UNREPLICABLE} BOOL;
		loc_Entf_NotbetriebBox2 : {REDUND_UNREPLICABLE} BOOL;
		loc_Entf_NotbetriebBox3 : {REDUND_UNREPLICABLE} BOOL;
		loc_Entf_NotbetriebBox4 : {REDUND_UNREPLICABLE} BOOL;
		loc_Entf_NotbetriebBox5 : {REDUND_UNREPLICABLE} BOOL;
		loc_Entf_NotbetriebBox6 : {REDUND_UNREPLICABLE} BOOL;
		loc_Sho_NotbetriebBox1 : {REDUND_UNREPLICABLE} BOOL;
		loc_Sho_NotbetriebBox2 : {REDUND_UNREPLICABLE} BOOL;
		loc_Sho_NotbetriebBox3 : {REDUND_UNREPLICABLE} BOOL;
		loc_Sho_NotbetriebBox4 : {REDUND_UNREPLICABLE} BOOL;
		loc_Sho_NotbetriebBox5 : {REDUND_UNREPLICABLE} BOOL;
		loc_Sho_NotbetriebBox6 : {REDUND_UNREPLICABLE} BOOL;
		loc_Wlo_NotbetriebBox1 : {REDUND_UNREPLICABLE} BOOL;
		loc_Wlo_NotbetriebBox2 : {REDUND_UNREPLICABLE} BOOL;
		loc_Wlo_NotbetriebBox3 : {REDUND_UNREPLICABLE} BOOL;
		loc_Wlo_NotbetriebBox4 : {REDUND_UNREPLICABLE} BOOL;
		loc_Wlo_NotbetriebBox5 : {REDUND_UNREPLICABLE} BOOL;
		loc_Wlo_NotbetriebBox6 : {REDUND_UNREPLICABLE} BOOL;
	END_VAR
END_FUNCTION_BLOCK

{REDUND_UNREPLICABLE} FUNCTION_BLOCK fbBoxenVentKlappen (*Funktionsbaustein für Ansteuerung Ventilatoren und Klappen*) (*$GROUP=User,$CAT=User,$GROUPICON=User.png,$CATICON=User.png*)
	VAR_INPUT
		Freigabe : {REDUND_UNREPLICABLE} BOOL;
		Ventilator1InBetrieb : {REDUND_UNREPLICABLE} BOOL;
		Ventilator2InBetrieb : {REDUND_UNREPLICABLE} BOOL;
		AnforderungVentilator1 : {REDUND_UNREPLICABLE} BOOL;
		AnforderungVentilator2 : {REDUND_UNREPLICABLE} BOOL;
		LuftaufbereitungInBetrieb : {REDUND_UNREPLICABLE} BOOL;
		DrzVent1UmschMitLuftaufb : {REDUND_UNREPLICABLE} REAL;
		DrzVent2UmschMitLuftaufb : {REDUND_UNREPLICABLE} REAL;
		DrehzahlVent1Umsch : {REDUND_UNREPLICABLE} REAL;
		DrehzahlVent2Umsch : {REDUND_UNREPLICABLE} REAL;
		DrehzahlVent1Betrieb : {REDUND_UNREPLICABLE} REAL;
		DrehzahlVent2Betrieb : {REDUND_UNREPLICABLE} REAL;
		DrehzahlVent1Min : {REDUND_UNREPLICABLE} REAL;
		DrehzahlVent1Max : {REDUND_UNREPLICABLE} REAL;
		DrehzahlVent2Min : {REDUND_UNREPLICABLE} REAL;
		DrehzahlVent2Max : {REDUND_UNREPLICABLE} REAL;
		RampeVent1Up : {REDUND_UNREPLICABLE} REAL;
		RampeVent1Down : {REDUND_UNREPLICABLE} REAL;
		RampeVent2Up : {REDUND_UNREPLICABLE} REAL;
		RampeVent2Down : {REDUND_UNREPLICABLE} REAL;
		BypassklappeOeffnen : {REDUND_UNREPLICABLE} BOOL;
		BypassklappeSchliessen : {REDUND_UNREPLICABLE} BOOL;
		Umschaltkl1Oeffnen : {REDUND_UNREPLICABLE} BOOL;
		Umschaltkl1Schliessen : {REDUND_UNREPLICABLE} BOOL;
		Umschaltkl2Oeffnen : {REDUND_UNREPLICABLE} BOOL;
		Umschaltkl2Schliessen : {REDUND_UNREPLICABLE} BOOL;
		Boxenklappe1Oeffnen : {REDUND_UNREPLICABLE} BOOL;
		Boxenklappe1Schliessen : {REDUND_UNREPLICABLE} BOOL;
		Boxenklappe2Oeffnen : {REDUND_UNREPLICABLE} BOOL;
		Boxenklappe2Schliessen : {REDUND_UNREPLICABLE} BOOL;
		Boxenklappe3Oeffnen : {REDUND_UNREPLICABLE} BOOL;
		Boxenklappe3Schliessen : {REDUND_UNREPLICABLE} BOOL;
		Boxenklappe4Oeffnen : {REDUND_UNREPLICABLE} BOOL;
		Boxenklappe4Schliessen : {REDUND_UNREPLICABLE} BOOL;
		Boxenklappe5Oeffnen : {REDUND_UNREPLICABLE} BOOL;
		Boxenklappe5Schliessen : {REDUND_UNREPLICABLE} BOOL;
		Boxenklappe6Oeffnen : {REDUND_UNREPLICABLE} BOOL;
		Boxenklappe6Schliessen : {REDUND_UNREPLICABLE} BOOL;
		EndlBypassGeschl : {REDUND_UNREPLICABLE} BOOL;
		EndlBypassOffen : {REDUND_UNREPLICABLE} BOOL;
		EndlUmschaltkl1Geschl : {REDUND_UNREPLICABLE} BOOL;
		EndlUmschaltkl1Offen : {REDUND_UNREPLICABLE} BOOL;
		EndlUmschaltkl2Geschl : {REDUND_UNREPLICABLE} BOOL;
		EndlUmschaltkl2Offen : {REDUND_UNREPLICABLE} BOOL;
		EndlBoxenklappe1Offen : {REDUND_UNREPLICABLE} BOOL;
		EndlBoxenklappe1Geschl : {REDUND_UNREPLICABLE} BOOL;
		EndlBoxenklappe2Offen : {REDUND_UNREPLICABLE} BOOL;
		EndlBoxenklappe2Geschl : {REDUND_UNREPLICABLE} BOOL;
		EndlBoxenklappe3Offen : {REDUND_UNREPLICABLE} BOOL;
		EndlBoxenklappe3Geschl : {REDUND_UNREPLICABLE} BOOL;
		EndlBoxenklappe4Offen : {REDUND_UNREPLICABLE} BOOL;
		EndlBoxenklappe4Geschl : {REDUND_UNREPLICABLE} BOOL;
		EndlBoxenklappe5Offen : {REDUND_UNREPLICABLE} BOOL;
		EndlBoxenklappe5Geschl : {REDUND_UNREPLICABLE} BOOL;
		EndlBoxenklappe6Offen : {REDUND_UNREPLICABLE} BOOL;
		EndlBoxenklappe6Geschl : {REDUND_UNREPLICABLE} BOOL;
		QuitFehler : {REDUND_UNREPLICABLE} BOOL;
		LaufzeitBypassklappe : {REDUND_UNREPLICABLE} UDINT;
		LaufzeitUmschaltklappe1 : {REDUND_UNREPLICABLE} UDINT;
		LaufzeitUmschaltklappe2 : {REDUND_UNREPLICABLE} UDINT;
		LaufzeitBoxenklappe1 : {REDUND_UNREPLICABLE} UDINT;
		LaufzeitBoxenklappe2 : {REDUND_UNREPLICABLE} UDINT;
		LaufzeitBoxenklappe3 : {REDUND_UNREPLICABLE} UDINT;
		LaufzeitBoxenklappe4 : {REDUND_UNREPLICABLE} UDINT;
		LaufzeitBoxenklappe5 : {REDUND_UNREPLICABLE} UDINT;
		LaufzeitBoxenklappe6 : {REDUND_UNREPLICABLE} UDINT;
		AnlaufverzZweiterVent : {REDUND_UNREPLICABLE} UDINT;
		Boxenklappe6Vorhanden : {REDUND_UNREPLICABLE} BOOL; (*True, wenn Boxenklappe in der Ausstattung vorhanden ist*)
		Boxenklappe5Vorhanden : {REDUND_UNREPLICABLE} BOOL; (*True, wenn Boxenklappe in der Ausstattung vorhanden ist*)
		Boxenklappe4Vorhanden : {REDUND_UNREPLICABLE} BOOL; (*True, wenn Boxenklappe in der Ausstattung vorhanden ist*)
		Boxenklappe3Vorhanden : {REDUND_UNREPLICABLE} BOOL; (*True, wenn Boxenklappe in der Ausstattung vorhanden ist*)
		Boxenklappe2Vorhanden : {REDUND_UNREPLICABLE} BOOL; (*True, wenn Boxenklappe in der Ausstattung vorhanden ist*)
		Boxenklappe1Vorhanden : {REDUND_UNREPLICABLE} BOOL; (*True, wenn Boxenklappe in der Ausstattung vorhanden ist*)
		UmluftklVonVent1Abhaengig : {REDUND_UNREPLICABLE} BOOL;
		UmluftklVonVent2Abhaengig : {REDUND_UNREPLICABLE} BOOL;
		Boxenkl1VonVent1Abhaengig : {REDUND_UNREPLICABLE} BOOL;
		Boxenkl1VonVent2Abhaengig : {REDUND_UNREPLICABLE} BOOL;
		Boxenkl2VonVent1Abhaengig : {REDUND_UNREPLICABLE} BOOL;
		Boxenkl2VonVent2Abhaengig : {REDUND_UNREPLICABLE} BOOL;
		Boxenkl3VonVent1Abhaengig : {REDUND_UNREPLICABLE} BOOL;
		Boxenkl3VonVent2Abhaengig : {REDUND_UNREPLICABLE} BOOL;
		Boxenkl4VonVent1Abhaengig : {REDUND_UNREPLICABLE} BOOL;
		Boxenkl4VonVent2Abhaengig : {REDUND_UNREPLICABLE} BOOL;
		Boxenkl5VonVent1Abhaengig : {REDUND_UNREPLICABLE} BOOL;
		Boxenkl5VonVent2Abhaengig : {REDUND_UNREPLICABLE} BOOL;
		Boxenkl6VonVent1Abhaengig : {REDUND_UNREPLICABLE} BOOL;
		Boxenkl6VonVent2Abhaengig : {REDUND_UNREPLICABLE} BOOL;
		BypassklVonVent1Abhaengig : {REDUND_UNREPLICABLE} BOOL;
		BypassklVonVent2Abhaengig : {REDUND_UNREPLICABLE} BOOL;
		EndlagenVhdBoxenklappe1 : {REDUND_UNREPLICABLE} BOOL; (*Sind keine Endlagen für die Klappe vorhanden, wird die Umschaltung der Klappe über die eingestellte Laufzeit simuliert*)
		EndlagenVhdBoxenklappe2 : {REDUND_UNREPLICABLE} BOOL; (*Sind keine Endlagen für die Klappe vorhanden, wird die Umschaltung der Klappe über die eingestellte Laufzeit simuliert*)
		EndlagenVhdBoxenklappe3 : {REDUND_UNREPLICABLE} BOOL; (*Sind keine Endlagen für die Klappe vorhanden, wird die Umschaltung der Klappe über die eingestellte Laufzeit simuliert*)
		EndlagenVhdBoxenklappe4 : {REDUND_UNREPLICABLE} BOOL; (*Sind keine Endlagen für die Klappe vorhanden, wird die Umschaltung der Klappe über die eingestellte Laufzeit simuliert*)
		EndlagenVhdBoxenklappe5 : {REDUND_UNREPLICABLE} BOOL; (*Sind keine Endlagen für die Klappe vorhanden, wird die Umschaltung der Klappe über die eingestellte Laufzeit simuliert*)
		EndlagenVhdBoxenklappe6 : {REDUND_UNREPLICABLE} BOOL; (*Sind keine Endlagen für die Klappe vorhanden, wird die Umschaltung der Klappe über die eingestellte Laufzeit simuliert*)
		EndlagenVhdUmschaltklappe1 : {REDUND_UNREPLICABLE} BOOL; (*Sind keine Endlagen für die Klappe vorhanden, wird die Umschaltung der Klappe über die eingestellte Laufzeit simuliert*)
		EndlagenVhdUmschaltklappe2 : {REDUND_UNREPLICABLE} BOOL; (*Sind keine Endlagen für die Klappe vorhanden, wird die Umschaltung der Klappe über die eingestellte Laufzeit simuliert*)
		EndlagenVhdBypassklappe : {REDUND_UNREPLICABLE} BOOL; (*Sind keine Endlagen für die Klappe vorhanden, wird die Umschaltung der Klappe über die eingestellte Laufzeit simuliert*)
	END_VAR
	VAR_OUTPUT
		FreigabeVentilator1Out : {REDUND_UNREPLICABLE} BOOL;
		FreigabeVentilator2Out : {REDUND_UNREPLICABLE} BOOL;
		DrehzahlVent1Out : {REDUND_UNREPLICABLE} REAL;
		DrehzahlVent2Out : {REDUND_UNREPLICABLE} REAL;
		BypassSchliessenOut : {REDUND_UNREPLICABLE} BOOL;
		BypassOeffnenOut : {REDUND_UNREPLICABLE} BOOL;
		Umschaltkl1SchliessenOut : {REDUND_UNREPLICABLE} BOOL;
		Umschaltkl1OeffnenOut : {REDUND_UNREPLICABLE} BOOL;
		Umschaltkl2SchliessenOut : {REDUND_UNREPLICABLE} BOOL;
		Umschaltkl2OeffnenOut : {REDUND_UNREPLICABLE} BOOL;
		Boxenklappe1OeffnenOut : {REDUND_UNREPLICABLE} BOOL;
		Boxenklappe1SchliessenOut : {REDUND_UNREPLICABLE} BOOL;
		Boxenklappe2OeffnenOut : {REDUND_UNREPLICABLE} BOOL;
		Boxenklappe2SchliessenOut : {REDUND_UNREPLICABLE} BOOL;
		Boxenklappe3OeffnenOut : {REDUND_UNREPLICABLE} BOOL;
		Boxenklappe3SchliessenOut : {REDUND_UNREPLICABLE} BOOL;
		Boxenklappe4OeffnenOut : {REDUND_UNREPLICABLE} BOOL;
		Boxenklappe4SchliessenOut : {REDUND_UNREPLICABLE} BOOL;
		Boxenklappe5OeffnenOut : {REDUND_UNREPLICABLE} BOOL;
		Boxenklappe5SchliessenOut : {REDUND_UNREPLICABLE} BOOL;
		Boxenklappe6OeffnenOut : {REDUND_UNREPLICABLE} BOOL;
		Boxenklappe6SchliessenOut : {REDUND_UNREPLICABLE} BOOL;
		UmschaltungAktiv : {REDUND_UNREPLICABLE} BOOL;
		FehlerLaufzeitBypass : {REDUND_UNREPLICABLE} BOOL;
		FehlerLaufzeitUmschaltkl1 : {REDUND_UNREPLICABLE} BOOL;
		FehlerLaufzeitUmschaltkl2 : {REDUND_UNREPLICABLE} BOOL;
		FehlerLaufzeitKlappeBox1 : {REDUND_UNREPLICABLE} BOOL;
		FehlerLaufzeitKlappeBox2 : {REDUND_UNREPLICABLE} BOOL;
		FehlerLaufzeitKlappeBox3 : {REDUND_UNREPLICABLE} BOOL;
		FehlerLaufzeitKlappeBox4 : {REDUND_UNREPLICABLE} BOOL;
		FehlerLaufzeitKlappeBox5 : {REDUND_UNREPLICABLE} BOOL;
		FehlerLaufzeitKlappeBox6 : {REDUND_UNREPLICABLE} BOOL;
		FehlerFuVentilator1 : {REDUND_UNREPLICABLE} BOOL;
		BypassklappeIstGeschl : {REDUND_UNREPLICABLE} BOOL; (*Statusausgang Stellung Klappe, wenn keine Endlagen vorhanden sind & Laufzeit <> 0 ist*)
		BypassklappeIstOffen : {REDUND_UNREPLICABLE} BOOL; (*Statusausgang Stellung Klappe, wenn keine Endlagen vorhanden sind & Laufzeit <> 0 ist*)
		Umschaltklappe1IstGeschl : {REDUND_UNREPLICABLE} BOOL; (*Statusausgang Stellung Klappe, wenn keine Endlagen vorhanden sind & Laufzeit <> 0 ist*)
		Umschaltklappe1IstOffen : {REDUND_UNREPLICABLE} BOOL; (*Statusausgang Stellung Klappe, wenn keine Endlagen vorhanden sind & Laufzeit <> 0 ist*)
		Umschaltklappe2IstGeschl : {REDUND_UNREPLICABLE} BOOL; (*Statusausgang Stellung Klappe, wenn keine Endlagen vorhanden sind & Laufzeit <> 0 ist*)
		Umschaltklappe2IstOffen : {REDUND_UNREPLICABLE} BOOL; (*Statusausgang Stellung Klappe, wenn keine Endlagen vorhanden sind & Laufzeit <> 0 ist*)
		Boxenklappe1IstOffen : {REDUND_UNREPLICABLE} BOOL; (*Statusausgang Stellung Klappe, wenn keine Endlagen vorhanden sind & Laufzeit <> 0 ist*)
		Boxenklappe1IstGeschl : {REDUND_UNREPLICABLE} BOOL; (*Statusausgang Stellung Klappe, wenn keine Endlagen vorhanden sind & Laufzeit <> 0 ist*)
		Boxenklappe2IstOffen : {REDUND_UNREPLICABLE} BOOL; (*Statusausgang Stellung Klappe, wenn keine Endlagen vorhanden sind & Laufzeit <> 0 ist*)
		Boxenklappe2IstGeschl : {REDUND_UNREPLICABLE} BOOL; (*Statusausgang Stellung Klappe, wenn keine Endlagen vorhanden sind & Laufzeit <> 0 ist*)
		Boxenklappe3IstOffen : {REDUND_UNREPLICABLE} BOOL; (*Statusausgang Stellung Klappe, wenn keine Endlagen vorhanden sind & Laufzeit <> 0 ist*)
		Boxenklappe3IstGeschl : {REDUND_UNREPLICABLE} BOOL; (*Statusausgang Stellung Klappe, wenn keine Endlagen vorhanden sind & Laufzeit <> 0 ist*)
		Boxenklappe4IstOffen : {REDUND_UNREPLICABLE} BOOL; (*Statusausgang Stellung Klappe, wenn keine Endlagen vorhanden sind & Laufzeit <> 0 ist*)
		Boxenklappe4IstGeschl : {REDUND_UNREPLICABLE} BOOL; (*Statusausgang Stellung Klappe, wenn keine Endlagen vorhanden sind & Laufzeit <> 0 ist*)
		Boxenklappe5IstOffen : {REDUND_UNREPLICABLE} BOOL; (*Statusausgang Stellung Klappe, wenn keine Endlagen vorhanden sind & Laufzeit <> 0 ist*)
		Boxenklappe5IstGeschl : {REDUND_UNREPLICABLE} BOOL; (*Statusausgang Stellung Klappe, wenn keine Endlagen vorhanden sind & Laufzeit <> 0 ist*)
		Boxenklappe6IstOffen : {REDUND_UNREPLICABLE} BOOL; (*Statusausgang Stellung Klappe, wenn keine Endlagen vorhanden sind & Laufzeit <> 0 ist*)
		Boxenklappe6IstGeschl : {REDUND_UNREPLICABLE} BOOL; (*Statusausgang Stellung Klappe, wenn keine Endlagen vorhanden sind & Laufzeit <> 0 ist*)
		FehlerFuVentilator2 : {REDUND_UNREPLICABLE} BOOL;
		curStep : {REDUND_UNREPLICABLE} USINT;
		RestAnlaufverzoegerung : {REDUND_UNREPLICABLE} UDINT;
		AnlaufverzVent1Aktiv : {REDUND_UNREPLICABLE} BOOL; (*Für Visu -> Ist TRUE, wenn Ventilator 1 angefordert und Anlaufverzögerung noch nicht abgelaufen ist*)
		AnlaufverzVent2Aktiv : {REDUND_UNREPLICABLE} BOOL; (*Für Visu -> Ist TRUE, wenn Ventilator 2 angefordert und Anlaufverzögerung noch nicht abgelaufen ist*)
	END_VAR
	VAR
		fbLascoEUhr_0 : {REDUND_UNREPLICABLE} fbLascoEUhr;
		fbLascoZdxx_0 : {REDUND_UNREPLICABLE} fbLascoZdxx;
		sekTick : {REDUND_UNREPLICABLE} BOOL;
		loc_AenderungBypassklappe : {REDUND_UNREPLICABLE} BOOL;
		loc_AenderungUmschaltklappe1 : {REDUND_UNREPLICABLE} BOOL;
		loc_AenderungUmschaltklappe2 : {REDUND_UNREPLICABLE} BOOL;
		loc_AenderungBoxenklappe1 : {REDUND_UNREPLICABLE} BOOL;
		loc_AenderungBoxenklappe2 : {REDUND_UNREPLICABLE} BOOL;
		loc_AenderungBoxenklappe3 : {REDUND_UNREPLICABLE} BOOL;
		loc_AenderungBoxenklappe4 : {REDUND_UNREPLICABLE} BOOL;
		loc_AenderungBoxenklappe5 : {REDUND_UNREPLICABLE} BOOL;
		loc_AenderungBoxenklappe6 : {REDUND_UNREPLICABLE} BOOL;
		loc_UmschaltungErforderlVent1 : {REDUND_UNREPLICABLE} BOOL;
		loc_UmschaltungErforderlVent2 : {REDUND_UNREPLICABLE} BOOL;
		fbFuVentilator1 : {REDUND_UNREPLICABLE} fbLascoFU;
		fbFuVentilator2 : {REDUND_UNREPLICABLE} fbLascoFU;
		Bypassklappe : {REDUND_UNREPLICABLE} fbBoxenKlappenanst;
		Umschaltklappe1 : {REDUND_UNREPLICABLE} fbBoxenKlappenanst;
		Umschaltklappe2 : {REDUND_UNREPLICABLE} fbBoxenKlappenanst;
		Boxenklappe1 : {REDUND_UNREPLICABLE} fbBoxenKlappenanst;
		Boxenklappe2 : {REDUND_UNREPLICABLE} fbBoxenKlappenanst;
		Boxenklappe3 : {REDUND_UNREPLICABLE} fbBoxenKlappenanst;
		Boxenklappe4 : {REDUND_UNREPLICABLE} fbBoxenKlappenanst;
		Boxenklappe5 : {REDUND_UNREPLICABLE} fbBoxenKlappenanst;
		Boxenklappe6 : {REDUND_UNREPLICABLE} fbBoxenKlappenanst;
		nextStep : {REDUND_UNREPLICABLE} USINT;
		stateEntry : {REDUND_UNREPLICABLE} BOOL;
		lastStep : {REDUND_UNREPLICABLE} USINT;
		TON_AnlaufverzVentilatoren : {REDUND_UNREPLICABLE} TON;
	END_VAR
END_FUNCTION_BLOCK

{REDUND_ERROR} {REDUND_UNREPLICABLE} FUNCTION_BLOCK fbBoxenKlappenanst (*Funktionsbaustein zur Ansteuerung von Klappen mit nur einem Wechsler-Relais (nicht angesteuert = Richtung A, angesteuert = Richtung B)*) (*$GROUP=User,$CAT=User,$GROUPICON=User.png,$CATICON=User.png*)
	VAR_INPUT
		Stoerung : {REDUND_UNREPLICABLE} BOOL;
		QuitFehler : {REDUND_UNREPLICABLE} BOOL;
		LaufzeitOeffnen : {REDUND_UNREPLICABLE} UDINT;
		LaufzeitSchliessen : {REDUND_UNREPLICABLE} UDINT;
		Oeffnen : {REDUND_UNREPLICABLE} BOOL;
		Schliessen : {REDUND_UNREPLICABLE} BOOL;
		EndlageOffen : {REDUND_UNREPLICABLE} BOOL;
		EndlageGeschl : {REDUND_UNREPLICABLE} BOOL;
		EndlagenVhd : {REDUND_UNREPLICABLE} BOOL; (*Wenn FALSE, wird die Umschaltung über die eingestellte Laufzeit simuliert und die Position der Klappe über "KlappeIstGeschl" bzw. "KlappeIstOffen" ausgegeben.*)
	END_VAR
	VAR_OUTPUT
		OeffnenOut : {REDUND_UNREPLICABLE} BOOL;
		SchliessenOut : {REDUND_UNREPLICABLE} BOOL;
		FehlerLaufzeitOeffnen : {REDUND_UNREPLICABLE} BOOL;
		FehlerLaufzeitSchliessen : {REDUND_UNREPLICABLE} BOOL;
		KlappeIstOffenOut : {REDUND_UNREPLICABLE} BOOL; (*Sind keine Endlagen vorhanden ("EndlagenVhd" ist FALSE), gibt der Ausgang die simulierte Position aus.*)
		KlappeIstGeschlOut : {REDUND_UNREPLICABLE} BOOL; (*Sind keine Endlagen vorhanden ("EndlagenVhd" ist FALSE), gibt der Ausgang die simulierte Position aus.*)
	END_VAR
	VAR
		step : {REDUND_UNREPLICABLE} USINT;
		stateEntry : {REDUND_UNREPLICABLE} BOOL;
		TON_Laufzeit : {REDUND_UNREPLICABLE} TON;
		TON_AnzVerz : {REDUND_UNREPLICABLE} TON;
	END_VAR
END_FUNCTION_BLOCK

{REDUND_ERROR} {REDUND_UNREPLICABLE} FUNCTION_BLOCK fbBoxenAbluftkl (*Funktionsbaustein zur Ansteuerung Abluftklappe/Abluftventilator*) (*$GROUP=User,$CAT=User,$GROUPICON=User.png,$CATICON=User.png*)
	VAR_INPUT
		Freigabe : {REDUND_UNREPLICABLE} BOOL;
		Quit : {REDUND_UNREPLICABLE} BOOL;
		Laufzeit : {REDUND_UNREPLICABLE} UDINT;
		Automatik : {REDUND_UNREPLICABLE} BOOL;
		AbluftFeuchteIst : {REDUND_UNREPLICABLE} REAL;
		Hysterese : {REDUND_UNREPLICABLE} REAL;
		AbluftFeuchteSoll : {REDUND_UNREPLICABLE} REAL;
		EndlageOffen : {REDUND_UNREPLICABLE} BOOL;
		EndlageGeschl : {REDUND_UNREPLICABLE} BOOL;
		Oeffnen : {REDUND_UNREPLICABLE} BOOL;
		Schliessen : {REDUND_UNREPLICABLE} BOOL;
	END_VAR
	VAR_OUTPUT
		OeffnenOut : {REDUND_UNREPLICABLE} BOOL;
		SchliessenOut : {REDUND_UNREPLICABLE} BOOL;
		FehlerLaufzeit : {REDUND_UNREPLICABLE} BOOL;
	END_VAR
	VAR
		stateEntry : {REDUND_UNREPLICABLE} BOOL;
		step : {REDUND_UNREPLICABLE} USINT;
		TON_Laufzeit : {REDUND_UNREPLICABLE} TON;
	END_VAR
END_FUNCTION_BLOCK

{REDUND_ERROR} {REDUND_UNREPLICABLE} FUNCTION_BLOCK fbBoxenAbluftvent (*Funktionsbaustein zur Ansteuerung Abluftventilator inkl. Drehzahlvorgabe*) (*$GROUP=User,$CAT=User,$GROUPICON=User.png,$CATICON=User.png*)
	VAR_INPUT
		Freigabe : {REDUND_UNREPLICABLE} BOOL;
		Automatik : {REDUND_UNREPLICABLE} BOOL;
		Ein : {REDUND_UNREPLICABLE} BOOL; (*Handbetrieb EIN*)
		VentilatorInBetrieb : {REDUND_UNREPLICABLE} BOOL;
		DrehzahlMin : {REDUND_UNREPLICABLE} REAL;
		DrehzahlMax : {REDUND_UNREPLICABLE} REAL;
		RampeUp : {REDUND_UNREPLICABLE} REAL;
		RampeDown : {REDUND_UNREPLICABLE} REAL;
		QuitFehler : {REDUND_UNREPLICABLE} BOOL;
		AbluftFeuchteIst : {REDUND_UNREPLICABLE} REAL;
		Hysterese : {REDUND_UNREPLICABLE} REAL;
		AbluftFeuchteSoll : {REDUND_UNREPLICABLE} REAL;
		DrehzahlSoll : {REDUND_UNREPLICABLE} REAL;
	END_VAR
	VAR_OUTPUT
		FehlerOut : {REDUND_UNREPLICABLE} BOOL;
		FreigabeVentilatorOut : {REDUND_UNREPLICABLE} BOOL;
		DrehzahlVentilatorOut : {REDUND_UNREPLICABLE} REAL;
	END_VAR
	VAR
		step : {REDUND_UNREPLICABLE} USINT;
		stateEntry : {REDUND_UNREPLICABLE} BOOL;
		fbFuAbluftventilator : {REDUND_UNREPLICABLE} fbLascoFU;
		sekTick : {REDUND_UNREPLICABLE} BOOL;
		fbLascoEUhr_0 : {REDUND_UNREPLICABLE} fbLascoEUhr;
		fbLascoZdxx_0 : {REDUND_UNREPLICABLE} fbLascoZdxx;
	END_VAR
END_FUNCTION_BLOCK

{REDUND_ERROR} {REDUND_UNREPLICABLE} FUNCTION_BLOCK fbBoxenUmschaltung (*Funktionsbaustein für Umschaltung Frischluft/Umluft*) (*$GROUP=User,$CAT=User,$GROUPICON=User.png,$CATICON=User.png*)
	VAR_INPUT
		AbluftTemp : {REDUND_UNREPLICABLE} REAL;
		SensorFrischluftVhd : {REDUND_UNREPLICABLE} BOOL;
		SensorDachluftVhd : {REDUND_UNREPLICABLE} BOOL;
		SensorAbluftVhd : {REDUND_UNREPLICABLE} BOOL;
		FrischluftTemp : {REDUND_UNREPLICABLE} REAL;
		DachluftTemp : {REDUND_UNREPLICABLE} REAL;
		DifferenzTempUmschaltung : {REDUND_UNREPLICABLE} REAL;
		FrischlDachlTempUmschaltung : {REDUND_UNREPLICABLE} REAL;
		Umschaltverz : {REDUND_UNREPLICABLE} UDINT;
		StatusSensorDachluftOk : {REDUND_UNREPLICABLE} BOOL;
		StatusSensorFrischluftOk : {REDUND_UNREPLICABLE} BOOL;
		StatusSensorAbluftOk : {REDUND_UNREPLICABLE} BOOL;
		Hysterese : {REDUND_UNREPLICABLE} REAL;
		Freigabe : {REDUND_UNREPLICABLE} BOOL;
	END_VAR
	VAR_OUTPUT
		FrischluftbetriebOut : {REDUND_UNREPLICABLE} BOOL;
		UmluftbetriebOut : {REDUND_UNREPLICABLE} BOOL;
	END_VAR
	VAR
		step : {REDUND_UNREPLICABLE} USINT;
		stateEntry : {REDUND_UNREPLICABLE} BOOL;
		TON_Umluft : {REDUND_UNREPLICABLE} TON;
		TON_Frischluft : {REDUND_UNREPLICABLE} TON;
		zzEdge00000 : {REDUND_UNREPLICABLE} BOOL;
		zzEdge00001 : {REDUND_UNREPLICABLE} BOOL;
		zzEdge00002 : {REDUND_UNREPLICABLE} BOOL;
		zzEdge00003 : {REDUND_UNREPLICABLE} BOOL;
		zzEdge00004 : {REDUND_UNREPLICABLE} BOOL;
		zzEdge00005 : {REDUND_UNREPLICABLE} BOOL;
		zzEdge00006 : {REDUND_UNREPLICABLE} BOOL;
		zzEdge00007 : {REDUND_UNREPLICABLE} BOOL;
	END_VAR
END_FUNCTION_BLOCK

{REDUND_ERROR} {REDUND_UNREPLICABLE} FUNCTION_BLOCK fbBoxenWLO (*Funktionsbaustein zur Ansteuerung Warmluftofen inkl. Solltemperatur-Vorgabe*) (*$GROUP=User,$CAT=User,$GROUPICON=User.png,$CATICON=User.png*)
	VAR_INPUT
		Freigabe : {REDUND_UNREPLICABLE} BOOL; (*Freigabe, wenn in Ausstattung vorhanden*)
		Automatikbetrieb : {REDUND_UNREPLICABLE} BOOL; (*Betriebsart Automatikbetrieb nach Aussenluft-Sättigungsdefizit*)
		Dauerbetrieb : {REDUND_UNREPLICABLE} BOOL; (*Betriebsart Dauerbetrieb*)
		FehlerSensorAussenluft : {REDUND_UNREPLICABLE} BOOL; (*Eingang Fehler Sensor Aussenluft (Automatikbetrieb nicht möglich)*)
		FrischluftSattDefizitIst : {REDUND_UNREPLICABLE} REAL;
		FrischluftSattDefizitSoll : {REDUND_UNREPLICABLE} REAL;
		Hysterese : {REDUND_UNREPLICABLE} REAL;
		UmschaltverzWitterung : {REDUND_UNREPLICABLE} UDINT;
		WarmlufttemperaturVorgabe : {REDUND_UNREPLICABLE} REAL;
		OptionBetriebsmldgVhd : {REDUND_UNREPLICABLE} BOOL;
		BetriebsmeldungWarmluftofen : {REDUND_UNREPLICABLE} BOOL;
		VerzBetriebsmeldung : {REDUND_UNREPLICABLE} UDINT;
		Auskuehlzeit : {REDUND_UNREPLICABLE} UDINT;
		QuitFehler : {REDUND_UNREPLICABLE} BOOL;
		WetterIstSchlecht : {REDUND_UNREPLICABLE} BOOL;
	END_VAR
	VAR_OUTPUT
		FreigabeWarmluftofenOut : {REDUND_UNREPLICABLE} BOOL;
		WarmlufttempSollOut : {REDUND_UNREPLICABLE} REAL;
		FehlerBetriebsmeldungOut : {REDUND_UNREPLICABLE} BOOL;
		FehlerSensorAussenluftOut : {REDUND_UNREPLICABLE} BOOL;
		WarmluftofenAktiv : {REDUND_UNREPLICABLE} BOOL; (*Warmluftofen aktiv (oder Nachkühlzeit nicht abgelaufen)*)
		RestAuskuehlzeit : {REDUND_UNREPLICABLE} UDINT;
	END_VAR
	VAR
		step : {REDUND_UNREPLICABLE} USINT;
		stateEntry : {REDUND_UNREPLICABLE} BOOL;
		TON_VerzBetriebsmeldung : {REDUND_UNREPLICABLE} TON;
		TOF_Auskuehlzeit : {REDUND_UNREPLICABLE} TOF;
		loc_WetterIstSchlecht : {REDUND_UNREPLICABLE} BOOL;
		loc_WetterIstGut : {REDUND_UNREPLICABLE} BOOL;
		zzEdge00000 : {REDUND_UNREPLICABLE} BOOL;
		zzEdge00001 : {REDUND_UNREPLICABLE} BOOL;
		TON_WetterIstGut : {REDUND_UNREPLICABLE} TON;
		TON_WetterIstSchlecht : {REDUND_UNREPLICABLE} TON;
	END_VAR
END_FUNCTION_BLOCK

{REDUND_ERROR} {REDUND_UNREPLICABLE} FUNCTION_BLOCK fbBoxenHeizreg (*Funktionsbaustein zur Ansteuerung eines Heizregisters inkl. Drehzahlvorgabe Heizungspumpe*) (*$GROUP=User,$CAT=User,$GROUPICON=User.png,$CATICON=User.png*)
	VAR_INPUT
		Freigabe : {REDUND_UNREPLICABLE} BOOL;
		QuitFehler : {REDUND_UNREPLICABLE} BOOL;
		DrehzahlHeizregisterSoll : {REDUND_UNREPLICABLE} REAL;
		Automatikbetrieb : {REDUND_UNREPLICABLE} BOOL;
		FehlerSensorAussenluft : {REDUND_UNREPLICABLE} BOOL;
		Dauerbetrieb : {REDUND_UNREPLICABLE} BOOL;
		FrischluftSattDefizitIst : {REDUND_UNREPLICABLE} REAL;
		FrischluftSattDefizitSoll : {REDUND_UNREPLICABLE} REAL;
		Hysterese : {REDUND_UNREPLICABLE} REAL;
		UmschaltverzWitterung : {REDUND_UNREPLICABLE} UDINT;
		WetterIstSchlecht : {REDUND_UNREPLICABLE} BOOL; (*Wird nur in für HB3000/HB4000 verwendet*)
	END_VAR
	VAR_OUTPUT
		FehlerOut : {REDUND_UNREPLICABLE} BOOL;
		FreigabeHeizregisterOut : {REDUND_UNREPLICABLE} BOOL;
		DrehzahlHeizregisterOut : {REDUND_UNREPLICABLE} REAL;
	END_VAR
	VAR
		zzEdge00000 : {REDUND_UNREPLICABLE} BOOL;
		zzEdge00001 : {REDUND_UNREPLICABLE} BOOL;
		step : {REDUND_UNREPLICABLE} USINT;
		stateEntry : {REDUND_UNREPLICABLE} BOOL;
		loc_WetterIstSchlecht : {REDUND_UNREPLICABLE} BOOL;
		loc_WetterIstGut : {REDUND_UNREPLICABLE} BOOL;
		TON_WetterIstGut : {REDUND_UNREPLICABLE} TON;
		TON_WetterIstSchlecht : {REDUND_UNREPLICABLE} TON;
	END_VAR
END_FUNCTION_BLOCK

{REDUND_ERROR} {REDUND_UNREPLICABLE} FUNCTION_BLOCK fbBoxenNotstrom (*Funktionsbaustein zur Ansteuerung eines Notstromaggregates inkl. Vorlaufzeit und Abfrage Betriebsmeldung*) (*$GROUP=User,$CAT=User,$GROUPICON=User.png,$CATICON=User.png*)
	VAR_INPUT
		Freigabe : {REDUND_UNREPLICABLE} BOOL;
		BetriebsmldgNotstromaggregat : {REDUND_UNREPLICABLE} BOOL;
		VerzBetriebsmeldung : {REDUND_UNREPLICABLE} UDINT;
		NotstromaggregatAngefordert : {REDUND_UNREPLICABLE} BOOL;
		QuitFehler : {REDUND_UNREPLICABLE} BOOL;
		Vorlaufzeit : {REDUND_UNREPLICABLE} UDINT;
		Nachlaufzeit : {REDUND_UNREPLICABLE} UDINT;
	END_VAR
	VAR_OUTPUT
		FreigabeNotstromaggregatOut : {REDUND_UNREPLICABLE} BOOL;
		FehlerOut : {REDUND_UNREPLICABLE} BOOL;
		NotstromBereitOut : {REDUND_UNREPLICABLE} BOOL;
		RestVorlaufzeit : {REDUND_UNREPLICABLE} UDINT;
		RestNachlaufzeit : {REDUND_UNREPLICABLE} UDINT;
	END_VAR
	VAR
		TON_VerzBetriebsmeldung : {REDUND_UNREPLICABLE} TON;
		TON_Vorlaufzeit : {REDUND_UNREPLICABLE} TON;
		TOF_Nachlaufzeit : {REDUND_UNREPLICABLE} TOF;
	END_VAR
END_FUNCTION_BLOCK

{REDUND_ERROR} {REDUND_UNREPLICABLE} FUNCTION_BLOCK fbBoxenSHO (*Funktionsbaustein Ansteuerung Scheitholzofen (Auskühlzeit)*) (*$GROUP=User,$CAT=User,$GROUPICON=User.png,$CATICON=User.png*)
	VAR_INPUT
		Freigabe : {REDUND_UNREPLICABLE} BOOL;
		Betriebsmeldung : {REDUND_UNREPLICABLE} BOOL;
		Auskuehlzeit : {REDUND_UNREPLICABLE} UDINT;
	END_VAR
	VAR_OUTPUT
		ScheitholzofenAktiv : {REDUND_UNREPLICABLE} BOOL;
		RestAuskuehlzeit : {REDUND_UNREPLICABLE} UDINT;
	END_VAR
	VAR
		TOF_Auskuehlzeit : {REDUND_UNREPLICABLE} TOF;
	END_VAR
END_FUNCTION_BLOCK

{REDUND_ERROR} {REDUND_UNREPLICABLE} FUNCTION_BLOCK fbBoxenLuftmengen (*Funktionsblock zur Ermittlung der erforderlichen Luftmengen für Ventilator 1&2 aus Boxenfläche*) (*$GROUP=User,$CAT=User,$GROUPICON=User.png,$CATICON=User.png*)
	VAR_INPUT
		Box1 : {REDUND_UNREPLICABLE} typBoxenLuftmengenIn;
		Box2 : {REDUND_UNREPLICABLE} typBoxenLuftmengenIn;
		Box3 : {REDUND_UNREPLICABLE} typBoxenLuftmengenIn;
		Box4 : {REDUND_UNREPLICABLE} typBoxenLuftmengenIn;
		Box5 : {REDUND_UNREPLICABLE} typBoxenLuftmengenIn;
		Box6 : {REDUND_UNREPLICABLE} typBoxenLuftmengenIn;
		LuftmengeSollProM2FrischlVent1 : {REDUND_UNREPLICABLE} REAL;
		LuftmengeSollProM2FrischlVent2 : {REDUND_UNREPLICABLE} REAL;
		LuftmengeSollProM2UmluftVent1 : {REDUND_UNREPLICABLE} REAL;
		LuftmengeSollProM2UmluftVent2 : {REDUND_UNREPLICABLE} REAL;
		RegisterflaecheEntfeuchter : {REDUND_UNREPLICABLE} REAL;
		LuftgeschwEntfeuchterMin : {REDUND_UNREPLICABLE} REAL;
		LuftgeschwEntfeuchterMax : {REDUND_UNREPLICABLE} REAL;
		FrischluftbetriebAktiv : {REDUND_UNREPLICABLE} BOOL;
		UmluftbetriebAktiv : {REDUND_UNREPLICABLE} BOOL;
		EntfeuchterInBetrieb : {REDUND_UNREPLICABLE} BOOL;
	END_VAR
	VAR_OUTPUT
		LuftmengeSollVent1Out : {REDUND_UNREPLICABLE} REAL;
		LuftmengeSollVent2Out : {REDUND_UNREPLICABLE} REAL;
	END_VAR
	VAR
		loc_LuftmengeSollVent1 : {REDUND_UNREPLICABLE} REAL;
		loc_LuftmengeSollVent2 : {REDUND_UNREPLICABLE} REAL;
		loc_MinLuftmengeMitEntfeuchter : {REDUND_UNREPLICABLE} REAL;
		loc_MaxLuftmengeMitEntfeuchter : {REDUND_UNREPLICABLE} REAL;
	END_VAR
END_FUNCTION_BLOCK

{REDUND_ERROR} {REDUND_UNREPLICABLE} FUNCTION_BLOCK fbRestzeit (*Funktionsbaustein zur Berechnung der Restzeit Lauf/Pause aus 24h Zeitfenstern (BOOL [24])*) (*$GROUP=User,$CAT=User,$GROUPICON=User.png,$CATICON=User.png*)
	VAR_INPUT
		Freigabe : {REDUND_UNREPLICABLE} BOOL;
		AktuelleStunde : {REDUND_UNREPLICABLE} USINT;
		AktuelleMinute : {REDUND_UNREPLICABLE} USINT;
		ZeitfensterIn : REFERENCE TO ARRAY[0..23] OF BOOL;
	END_VAR
	VAR_OUTPUT
		ZeitfensterAktiv : {REDUND_UNREPLICABLE} BOOL;
		RestzeitStundenOut : {REDUND_UNREPLICABLE} UINT;
		RestzeitMinutenOut : {REDUND_UNREPLICABLE} UINT;
	END_VAR
	VAR
		loc_MinutenRestTag : {REDUND_UNREPLICABLE} UINT;
		loc_Aenderung : {REDUND_UNREPLICABLE} DINT;
		MEM_ZeitfensterIn : {REDUND_UNREPLICABLE} BOOL;
		loc_firstInitLauf : {REDUND_UNREPLICABLE} BOOL;
		i : {REDUND_UNREPLICABLE} USINT;
		loc_StundeEndeZeitfTag : {REDUND_UNREPLICABLE} USINT;
		loc_MinutenRestFolgetag : {REDUND_UNREPLICABLE} UINT;
		ii : {REDUND_UNREPLICABLE} USINT;
		loc_StundeEndeZeitfFolgetag : {REDUND_UNREPLICABLE} USINT;
		loc_MinutenRestGesamt : {REDUND_UNREPLICABLE} UINT;
		loc_firstInitPause : {REDUND_UNREPLICABLE} BOOL;
		loc_RestzeitStunden : {REDUND_UNREPLICABLE} UINT;
	END_VAR
END_FUNCTION_BLOCK
```
